gfCNCPoint3[18033] = {X 35.8445, Y 45.9080, Z -4.6667, A 0.000, B 0.000, C 0.000 }
gfCNCPoint3[18034] = {X 35.7593, Y 45.0000, Z -4.6667, A 0.000, B 0.000, C 0.000 }
gfCNCPoint3[18035] = {X 35.7593, Y 44.7148, Z -4.6667, A 0.000, B 0.000, C 0.000 }
gfCNCPoint3[18036] = {X 36.2393, Y 44.7148, Z -4.6667, A 0.000, B 0.000, C 0.000 }
gfCNCPoint3[18037] = {X 36.2397, Y 44.1483, Z -4.6667, A 0.000, B 0.000, C 0.000 }
gfCNCPoint3[18038] = {X 36.3680, Y 43.1522, Z -4.6667, A 0.000, B 0.000, C 0.000 }
gfCNCPoint3[18039] = {X 36.7189, Y 42.2112, Z -4.6667, A 0.000, B 0.000, C 0.000 }
gfCNCPoint3[18040] = {X 37.2740, Y 41.3742, Z -4.6667, A 0.000, B 0.000, C 0.000 }
gfCNCPoint3[18041] = {X 38.0044, Y 40.6849, Z -4.6667, A 0.000, B 0.000, C 0.000 }
gfCNCPoint3[18042] = {X 38.8721, Y 40.1793, Z -4.6667, A 0.000, B 0.000, C 0.000 }
gfCNCPoint3[18043] = {X 39.4558, Y 38.7988, Z -4.6667, A 0.000, B 0.000, C 0.000 }
gfCNCPoint3[18044] = {X 39.9904, Y 37.3987, Z -4.6667, A 0.000, B 0.000, C 0.000 }
gfCNCPoint3[18045] = {X 48.2011, Y 15.3544, Z -4.6667, A 0.000, B 0.000, C 0.000 }
gfCNCPoint3[18046] = {X 47.8187, Y 14.6115, Z -4.6667, A 0.000, B 0.000, C 0.000 }
gfCNCPoint3[18047] = {X 47.5835, Y 13.8097, Z -4.6667, A 0.000, B 0.000, C 0.000 }
gfCNCPoint3[18048] = {X 47.5042, Y 12.9779, Z -4.6667, A 0.000, B 0.000, C 0.000 }
gfCNCPoint3[18049] = {X 47.5042, Y 12.1868, Z -4.6667, A 0.000, B 0.000, C 0.000 }
gfCNCPoint3[18050] = {X 47.6145, Y 11.2077, Z -4.6667, A 0.000, B 0.000, C 0.000 }
gfCNCPoint3[18051] = {X 47.9400, Y 10.2777, Z -4.6667, A 0.000, B 0.000, C 0.000 }
gfCNCPoint3[18052] = {X 48.4642, Y 9.4435, Z -4.6667, A 0.000, B 0.000, C 0.000 }
gfCNCPoint3[18053] = {X 49.1609, Y 8.7468, Z -4.6667, A 0.000, B 0.000, C 0.000 }
gfCNCPoint3[18054] = {X 49.9951, Y 8.2226, Z -4.6667, A 0.000, B 0.000, C 0.000 }
gfCNCPoint3[18055] = {X 50.9251, Y 7.8971, Z -4.6667, A 0.000, B 0.000, C 0.000 }
gfCNCPoint3[18056] = {X 51.9042, Y 7.7868, Z -4.6667, A 0.000, B 0.000, C 0.000 }
gfCNCPoint3[18057] = {X 59.6221, Y 7.7868, Z -4.6667, A 0.000, B 0.000, C 0.000 }
gfCNCPoint3[18058] = {X 60.6012, Y 7.8971, Z -4.6667, A 0.000, B 0.000, C 0.000 }
gfCNCPoint3[18059] = {X 61.5312, Y 8.2226, Z -4.6667, A 0.000, B 0.000, C 0.000 }
gfCNCPoint3[18060] = {X 62.3655, Y 8.7468, Z -4.6667, A 0.000, B 0.000, C 0.000 }
gfCNCPoint3[18061] = {X 63.0622, Y 9.4435, Z -4.6667, A 0.000, B 0.000, C 0.000 }
gfCNCPoint3[18062] = {X 63.5864, Y 10.2777, Z -4.6667, A 0.000, B 0.000, C 0.000 }
gfCNCPoint3[18063] = {X 63.9118, Y 11.2077, Z -4.6667, A 0.000, B 0.000, C 0.000 }
gfCNCPoint3[18064] = {X 64.0221, Y 12.1868, Z -4.6667, A 0.000, B 0.000, C 0.000 }
gfCNCPoint3[18065] = {X 64.0219, Y 13.0233, Z -4.6667, A 0.000, B 0.000, C 0.000 }
gfCNCPoint3[18066] = {X 63.9336, Y 13.8563, Z -4.6667, A 0.000, B 0.000, C 0.000 }
gfCNCPoint3[18067] = {X 63.6890, Y 14.6575, Z -4.6667, A 0.000, B 0.000, C 0.000 }
gfCNCPoint3[18068] = {X 63.2970, Y 15.3978, Z -4.6667, A 0.000, B 0.000, C 0.000 }
gfCNCPoint3[18069] = {X 63.5008, Y 15.9354, Z -4.6667, A 0.000, B 0.000, C 0.000 }
gfCNCPoint3[18070] = {X 66.3154, Y 23.4040, Z -4.6667, A 0.000, B 0.000, C 0.000 }
gfCNCPoint3[18071] = {X 72.2844, Y 39.4717, Z -4.6667, A 0.000, B 0.000, C 0.000 }
gfCNCPoint3[18072] = {X 72.5774, Y 40.2087, Z -4.6667, A 0.000, B 0.000, C 0.000 }
gfCNCPoint3[18073] = {X 73.4349, Y 40.7272, Z -4.6667, A 0.000, B 0.000, C 0.000 }
gfCNCPoint3[18074] = {X 74.1528, Y 41.4262, Z -4.6667, A 0.000, B 0.000, C 0.000 }
gfCNCPoint3[18075] = {X 74.6940, Y 42.2695, Z -4.6667, A 0.000, B 0.000, C 0.000 }
gfCNCPoint3[18076] = {X 75.0304, Y 43.2134, Z -4.6667, A 0.000, B 0.000, C 0.000 }
gfCNCPoint3[18077] = {X 75.1445, Y 44.2089, Z -4.6667, A 0.000, B 0.000, C 0.000 }
gfCNCPoint3[18078] = {X 75.1445, Y 45.0000, Z -4.6667, A 0.000, B 0.000, C 0.000 }
gfCNCPoint3[18079] = {X 75.0341, Y 45.9791, Z -4.6667, A 0.000, B 0.000, C 0.000 }
gfCNCPoint3[18080] = {X 74.7087, Y 46.9091, Z -4.6667, A 0.000, B 0.000, C 0.000 }
gfCNCPoint3[18081] = {X 74.1845, Y 47.7434, Z -4.6667, A 0.000, B 0.000, C 0.000 }
gfCNCPoint3[18082] = {X 73.4878, Y 48.4401, Z -4.6667, A 0.000, B 0.000, C 0.000 }
gfCNCPoint3[18083] = {X 72.6535, Y 48.9643, Z -4.6667, A 0.000, B 0.000, C 0.000 }
gfCNCPoint3[18084] = {X 71.7236, Y 49.2897, Z -4.6667, A 0.000, B 0.000, C 0.000 }
gfCNCPoint3[18085] = {X 70.7445, Y 49.4000, Z -4.6667, A 0.000, B 0.000, C 0.000 }
gfCNCPoint3[18086] = {X 64.1851, Y 49.4000, Z -4.6667, A 0.000, B 0.000, C 0.000 }
gfCNCPoint3[18087] = {X 63.2060, Y 49.2897, Z -4.6667, A 0.000, B 0.000, C 0.000 }
gfCNCPoint3[18088] = {X 62.2760, Y 48.9643, Z -4.6667, A 0.000, B 0.000, C 0.000 }
gfCNCPoint3[18089] = {X 61.4418, Y 48.4401, Z -4.6667, A 0.000, B 0.000, C 0.000 }
gfCNCPoint3[18090] = {X 60.7451, Y 47.7434, Z -4.6667, A 0.000, B 0.000, C 0.000 }
gfCNCPoint3[18091] = {X 60.2209, Y 46.9091, Z -4.6667, A 0.000, B 0.000, C 0.000 }
gfCNCPoint3[18092] = {X 59.8955, Y 45.9791, Z -4.6667, A 0.000, B 0.000, C 0.000 }
gfCNCPoint3[18093] = {X 59.7851, Y 45.0000, Z -4.6667, A 0.000, B 0.000, C 0.000 }
gfCNCPoint3[18094] = {X 59.7856, Y 44.1483, Z -4.6667, A 0.000, B 0.000, C 0.000 }
gfCNCPoint3[18095] = {X 59.8784, Y 43.3079, Z -4.6667, A 0.000, B 0.000, C 0.000 }
gfCNCPoint3[18096] = {X 60.1302, Y 42.5007, Z -4.6667, A 0.000, B 0.000, C 0.000 }
gfCNCPoint3[18097] = {X 60.5318, Y 41.7567, Z -4.6667, A 0.000, B 0.000, C 0.000 }
gfCNCPoint3[18098] = {X 59.9510, Y 40.1692, Z -4.6667, A 0.000, B 0.000, C 0.000 }
gfCNCPoint3[18099] = {X 52.1329, Y 40.1692, Z -4.6667, A 0.000, B 0.000, C 0.000 }
gfCNCPoint3[18100] = {X 51.4225, Y 42.0778, Z -4.6667, A 0.000, B 0.000, C 0.000 }
gfCNCPoint3[18101] = {X 51.7254, Y 42.7537, Z -4.6667, A 0.000, B 0.000, C 0.000 }
gfCNCPoint3[18102] = {X 51.9106, Y 43.4709, Z -4.6667, A 0.000, B 0.000, C 0.000 }
gfCNCPoint3[18103] = {X 51.9729, Y 44.2089, Z -4.6667, A 0.000, B 0.000, C 0.000 }
gfCNCPoint3[18104] = {X 51.9729, Y 45.0000, Z -4.6667, A 0.000, B 0.000, C 0.000 }
gfCNCPoint3[18105] = {X 51.8626, Y 45.9791, Z -4.6667, A 0.000, B 0.000, C 0.000 }
gfCNCPoint3[18106] = {X 51.5372, Y 46.9091, Z -4.6667, A 0.000, B 0.000, C 0.000 }
gfCNCPoint3[18107] = {X 51.0130, Y 47.7434, Z -4.6667, A 0.000, B 0.000, C 0.000 }
gfCNCPoint3[18108] = {X 50.3163, Y 48.4401, Z -4.6667, A 0.000, B 0.000, C 0.000 }
gfCNCPoint3[18109] = {X 49.4820, Y 48.9643, Z -4.6667, A 0.000, B 0.000, C 0.000 }
gfCNCPoint3[18110] = {X 48.5520, Y 49.2897, Z -4.6667, A 0.000, B 0.000, C 0.000 }
gfCNCPoint3[18111] = {X 47.5729, Y 49.4000, Z -4.6667, A 0.000, B 0.000, C 0.000 }
gfCNCPoint3[18112] = {X 40.6393, Y 49.4000, Z -4.6667, A 0.000, B 0.000, C 0.000 }
gfCNCPoint3[18113] = {X 39.6602, Y 49.2897, Z -4.6667, A 0.000, B 0.000, C 0.000 }
gfCNCPoint3[18114] = {X 38.7302, Y 48.9643, Z -4.6667, A 0.000, B 0.000, C 0.000 }
gfCNCPoint3[18115] = {X 37.8959, Y 48.4401, Z -4.6667, A 0.000, B 0.000, C 0.000 }
gfCNCPoint3[18116] = {X 37.1992, Y 47.7434, Z -4.6667, A 0.000, B 0.000, C 0.000 }
gfCNCPoint3[18117] = {X 36.6750, Y 46.9091, Z -4.6667, A 0.000, B 0.000, C 0.000 }
gfCNCPoint3[18118] = {X 36.3496, Y 45.9791, Z -4.6667, A 0.000, B 0.000, C 0.000 }
gfCNCPoint3[18119] = {X 36.2393, Y 45.0000, Z -4.6667, A 0.000, B 0.000, C 0.000 }
gfCNCPoint3[18120] = {X 36.2393, Y 44.7148, Z -4.6667, A 0.000, B 0.000, C 0.000 }
gfCNCPoint3[18121] = {X 35.7593, Y 44.7148, Z -4.6667, A 0.000, B 0.000, C 0.000 }
gfCNCPoint3[18122] = {X 35.2211, Y 46.0074, Z -4.6667, A 0.000, B 0.000, C 0.000 }
gfCNCPoint3[18123] = {X 34.4930, Y 47.2034, Z -4.6667, A 0.000, B 0.000, C 0.000 }
gfCNCPoint3[18124] = {X 33.5918, Y 48.2750, Z -4.6667, A 0.000, B 0.000, C 0.000 }
gfCNCPoint3[18125] = {X 33.2092, Y 48.6435, Z -4.6667, A 0.000, B 0.000, C 0.000 }
gfCNCPoint3[18126] = {X 32.8060, Y 48.9892, Z -4.6667, A 0.000, B 0.000, C 0.000 }
gfCNCPoint3[18127] = {X 32.2679, Y 49.4243, Z -4.6667, A 0.000, B 0.000, C 0.000 }
gfCNCPoint3[18128] = {X 31.1814, Y 50.1797, Z -4.6667, A 0.000, B 0.000, C 0.000 }
gfCNCPoint3[18129] = {X 29.9980, Y 50.7716, Z -4.6667, A 0.000, B 0.000, C 0.000 }
gfCNCPoint3[18130] = {X 28.7420, Y 51.1880, Z -4.6667, A 0.000, B 0.000, C 0.000 }
gfCNCPoint3[18131] = {X 27.4393, Y 51.4201, Z -4.6667, A 0.000, B 0.000, C 0.000 }
gfCNCPoint3[18132] = {X 26.1168, Y 51.4633, Z -4.6667, A 0.000, B 0.000, C 0.000 }
gfCNCPoint3[18133] = {X 23.6796, Y 52.5818, Z -4.6667, A 0.000, B 0.000, C 0.000 }
gfCNCPoint3[18134] = {X 21.1619, Y 53.5051, Z -4.6667, A 0.000, B 0.000, C 0.000 }
gfCNCPoint3[18135] = {X 18.9497, Y 54.1342, Z -4.6667, A 0.000, B 0.000, C 0.000 }
gfCNCPoint3[18136] = {X 16.6929, Y 54.5773, Z -4.6667, A 0.000, B 0.000, C 0.000 }
gfCNCPoint3[18137] = {X 14.4071, Y 54.8314, Z -4.6667, A 0.000, B 0.000, C 0.000 }
gfCNCPoint3[18138] = {X 12.1081, Y 54.8947, Z -4.6667, A 0.000, B 0.000, C 0.000 }
gfCNCPoint3[18139] = {X 9.8118, Y 54.7667, Z -4.6667, A 0.000, B 0.000, C 0.000 }
gfCNCPoint3[18140] = {X 7.5341, Y 54.4485, Z -4.6667, A 0.000, B 0.000, C 0.000 }
gfCNCPoint3[18141] = {X 7.1099, Y 54.3677, Z -4.6667, A 0.000, B 0.000, C 0.000 }
gfCNCPoint3[18142] = {X 6.6870, Y 54.2803, Z -4.6667, A 0.000, B 0.000, C 0.000 }
gfCNCPoint3[18143] = {X 5.6890, Y 54.0441, Z -4.6667, A 0.000, B 0.000, C 0.000 }
gfCNCPoint3[18144] = {X 4.7034, Y 53.7607, Z -4.6667, A 0.000, B 0.000, C 0.000 }
gfCNCPoint3[18145] = {X 4.7034, Y 95.2950, Z -4.6667, A 0.000, B 0.000, C 0.000 }
gfCNCPoint3[18146] = {X 117.9387, Y 95.2950, Z -4.6667, A 0.000, B 0.000, C 0.000 }
gfCNCPoint3[18147] = {X 118.3612, Y 94.0786, Z -4.6667, A 0.000, B 0.000, C 0.000 }
gfCNCPoint3[18148] = {X 118.9914, Y 92.9556, Z -4.6667, A 0.000, B 0.000, C 0.000 }
gfCNCPoint3[18149] = {X 119.8096, Y 91.9613, Z -4.6667, A 0.000, B 0.000, C 0.000 }
gfCNCPoint3[18150] = {X 120.7902, Y 91.1266, Z -4.6667, A 0.000, B 0.000, C 0.000 }
gfCNCPoint3[18151] = {X 121.9025, Y 90.4778, Z -4.6667, A 0.000, B 0.000, C 0.000 }
gfCNCPoint3[18152] = {X 123.1117, Y 90.0351, Z -4.6667, A 0.000, B 0.000, C 0.000 }
gfCNCPoint3[18153] = {X 124.3800, Y 89.8124, Z -4.6667, A 0.000, B 0.000, C 0.000 }
gfCNCPoint3[18154] = {X 125.0501, Y 89.7112, Z -4.6667, A 0.000, B 0.000, C 0.000 }
gfCNCPoint3[18155] = {X 125.3582, Y 89.6652, Z -4.6667, A 0.000, B 0.000, C 0.000 }
gfCNCPoint3[18156] = {X 125.6646, Y 89.6090, Z -4.6667, A 0.000, B 0.000, C 0.000 }
gfCNCPoint3[18157] = {X 126.4915, Y 88.7984, Z -4.6667, A 0.000, B 0.000, C 0.000 }
gfCNCPoint3[18158] = {X 127.2841, Y 87.9542, Z -4.6667, A 0.000, B 0.000, C 0.000 }
gfCNCPoint3[18159] = {X 152.2076, Y 60.5847, Z -4.6667, A 0.000, B 0.000, C 0.000 }
gfCNCPoint3[18160] = {X 152.0684, Y 59.7898, Z -4.6667, A 0.000, B 0.000, C 0.000 }
gfCNCPoint3[18161] = {X 152.0181, Y 58.9845, Z -4.6667, A 0.000, B 0.000, C 0.000 }
gfCNCPoint3[18162] = {X 152.0180, Y 58.0000, Z -4.6667, A 0.000, B 0.000, C 0.000 }
gfCNCPoint3[18163] = {X 152.1286, Y 56.7358, Z -4.6667, A 0.000, B 0.000, C 0.000 }
gfCNCPoint3[18164] = {X 152.4570, Y 55.5101, Z -4.6667, A 0.000, B 0.000, C 0.000 }
gfCNCPoint3[18165] = {X 152.9933, Y 54.3600, Z -4.6667, A 0.000, B 0.000, C 0.000 }
gfCNCPoint3[18166] = {X 153.7212, Y 53.3205, Z -4.6667, A 0.000, B 0.000, C 0.000 }
gfCNCPoint3[18167] = {X 154.6185, Y 52.4232, Z -4.6667, A 0.000, B 0.000, C 0.000 }
gfCNCPoint3[18168] = {X 155.6580, Y 51.6953, Z -4.6667, A 0.000, B 0.000, C 0.000 }
gfCNCPoint3[18169] = {X 156.8081, Y 51.1590, Z -4.6667, A 0.000, B 0.000, C 0.000 }
gfCNCPoint3[18170] = {X 158.0338, Y 50.8306, Z -4.6667, A 0.000, B 0.000, C 0.000 }
gfCNCPoint3[18171] = {X 159.2980, Y 50.7200, Z -4.6667, A 0.000, B 0.000, C 0.000 }
gfCNCPoint3[18172] = {X 178.5335, Y 50.7200, Z -4.6667, A 0.000, B 0.000, C 0.000 }
gfCNCPoint3[18173] = {X 179.7870, Y 50.8287, Z -4.6667, A 0.000, B 0.000, C 0.000 }
gfCNCPoint3[18174] = {X 181.0031, Y 51.1517, Z -4.6667, A 0.000, B 0.000, C 0.000 }
gfCNCPoint3[18175] = {X 182.1454, Y 51.6792, Z -4.6667, A 0.000, B 0.000, C 0.000 }
gfCNCPoint3[18176] = {X 183.1798, Y 52.3955, Z -4.6667, A 0.000, B 0.000, C 0.000 }
gfCNCPoint3[18177] = {X 184.0880, Y 53.2941, Z -4.6667, A 0.000, B 0.000, C 0.000 }
gfCNCPoint3[18178] = {X 184.8252, Y 54.3376, Z -4.6667, A 0.000, B 0.000, C 0.000 }
gfCNCPoint3[18179] = {X 185.3685, Y 55.4939, Z -4.6667, A 0.000, B 0.000, C 0.000 }
gfCNCPoint3[18180] = {X 185.7014, Y 56.7273, Z -4.6667, A 0.000, B 0.000, C 0.000 }
gfCNCPoint3[18181] = {X 185.8135, Y 58.0000, Z -4.6667, A 0.000, B 0.000, C 0.000 }
gfCNCPoint3[18182] = {X 185.8133, Y 58.9942, Z -4.6667, A 0.000, B 0.000, C 0.000 }
gfCNCPoint3[18183] = {X 185.7648, Y 59.7749, Z -4.6667, A 0.000, B 0.000, C 0.000 }
gfCNCPoint3[18184] = {X 185.6328, Y 60.5459, Z -4.6667, A 0.000, B 0.000, C 0.000 }
gfCNCPoint3[18185] = {X 211.6613, Y 88.9545, Z -4.6667, A 0.000, B 0.000, C 0.000 }
gfCNCPoint3[18186] = {X 212.0333, Y 89.3391, Z -4.6667, A 0.000, B 0.000, C 0.000 }
gfCNCPoint3[18187] = {X 212.4256, Y 89.7031, Z -4.6667, A 0.000, B 0.000, C 0.000 }
gfCNCPoint3[18188] = {X 212.6034, Y 89.7411, Z -4.6667, A 0.000, B 0.000, C 0.000 }
gfCNCPoint3[18189] = {X 213.4473, Y 89.8474, Z -4.6667, A 0.000, B 0.000, C 0.000 }
gfCNCPoint3[18190] = {X 214.4298, Y 89.7705, Z -4.6667, A 0.000, B 0.000, C 0.000 }
gfCNCPoint3[18191] = {X 215.4138, Y 89.7168, Z -4.6667, A 0.000, B 0.000, C 0.000 }
gfCNCPoint3[18192] = {X 215.6261, Y 89.6935, Z -4.6667, A 0.000, B 0.000, C 0.000 }
gfCNCPoint3[18193] = {X 215.8213, Y 89.6066, Z -4.6667, A 0.000, B 0.000, C 0.000 }
gfCNCPoint3[18194] = {X 239.3462, Y 74.5356, Z -4.6667, A 0.000, B 0.000, C 0.000 }
gfCNCPoint3[18195] = {X 220.5436, Y 67.1569, Z -4.6667, A 0.000, B 0.000, C 0.000 }
gfCNCPoint3[18196] = {X 219.0950, Y 66.6707, Z -4.6667, A 0.000, B 0.000, C 0.000 }
gfCNCPoint3[18197] = {X 217.6003, Y 66.3535, Z -4.6667, A 0.000, B 0.000, C 0.000 }
gfCNCPoint3[18198] = {X 216.0790, Y 66.2097, Z -4.6667, A 0.000, B 0.000, C 0.000 }
gfCNCPoint3[18199] = {X 214.8523, Y 66.0623, Z -4.6667, A 0.000, B 0.000, C 0.000 }
gfCNCPoint3[18200] = {X 213.6682, Y 65.7097, Z -4.6667, A 0.000, B 0.000, C 0.000 }
gfCNCPoint3[18201] = {X 212.5607, Y 65.1618, Z -4.6667, A 0.000, B 0.000, C 0.000 }
gfCNCPoint3[18202] = {X 211.5619, Y 64.4346, Z -4.6667, A 0.000, B 0.000, C 0.000 }
gfCNCPoint3[18203] = {X 210.7004, Y 63.5490, Z -4.6667, A 0.000, B 0.000, C 0.000 }
gfCNCPoint3[18204] = {X 210.0011, Y 62.5304, Z -4.6667, A 0.000, B 0.000, C 0.000 }
gfCNCPoint3[18205] = {X 209.4841, Y 61.4082, Z -4.6667, A 0.000, B 0.000, C 0.000 }
gfCNCPoint3[18206] = {X 209.1643, Y 60.2148, Z -4.6667, A 0.000, B 0.000, C 0.000 }
gfCNCPoint3[18207] = {X 209.0510, Y 58.9845, Z -4.6667, A 0.000, B 0.000, C 0.000 }
gfCNCPoint3[18208] = {X 209.0508, Y 58.0000, Z -4.6667, A 0.000, B 0.000, C 0.000 }
gfCNCPoint3[18209] = {X 209.1477, Y 56.8162, Z -4.6667, A 0.000, B 0.000, C 0.000 }
gfCNCPoint3[18210] = {X 209.4358, Y 55.6638, Z -4.6667, A 0.000, B 0.000, C 0.000 }
gfCNCPoint3[18211] = {X 209.9075, Y 54.5737, Z -4.6667, A 0.000, B 0.000, C 0.000 }
gfCNCPoint3[18212] = {X 210.5502, Y 53.5748, Z -4.6667, A 0.000, B 0.000, C 0.000 }
gfCNCPoint3[18213] = {X 211.3467, Y 52.6937, Z -4.6667, A 0.000, B 0.000, C 0.000 }
gfCNCPoint3[18214] = {X 212.2759, Y 51.9538, Z -4.6667, A 0.000, B 0.000, C 0.000 }
gfCNCPoint3[18215] = {X 213.3131, Y 51.3749, Z -4.6667, A 0.000, B 0.000, C 0.000 }
gfCNCPoint3[18216] = {X 214.4306, Y 50.9724, Z -4.6667, A 0.000, B 0.000, C 0.000 }
gfCNCPoint3[18217] = {X 215.3724, Y 50.7834, Z -4.6667, A 0.000, B 0.000, C 0.000 }
gfCNCPoint3[18218] = {X 216.3308, Y 50.7200, Z -4.6667, A 0.000, B 0.000, C 0.000 }
gfCNCPoint3[18219] = {X 237.2617, Y 50.7200, Z -4.6667, A 0.000, B 0.000, C 0.000 }
gfCNCPoint3[18220] = {X 238.3057, Y 50.7953, Z -4.6667, A 0.000, B 0.000, C 0.000 }
gfCNCPoint3[18221] = {X 239.3282, Y 51.0195, Z -4.6667, A 0.000, B 0.000, C 0.000 }
gfCNCPoint3[18222] = {X 240.3080, Y 51.3880, Z -4.6667, A 0.000, B 0.000, C 0.000 }
gfCNCPoint3[18223] = {X 241.2247, Y 51.8932, Z -4.6667, A 0.000, B 0.000, C 0.000 }
gfCNCPoint3[18224] = {X 242.0741, Y 52.5375, Z -4.6667, A 0.000, B 0.000, C 0.000 }
gfCNCPoint3[18225] = {X 242.8203, Y 53.2989, Z -4.6667, A 0.000, B 0.000, C 0.000 }
gfCNCPoint3[18226] = {X 243.4473, Y 54.1611, Z -4.6667, A 0.000, B 0.000, C 0.000 }
gfCNCPoint3[18227] = {X 243.9416, Y 55.1057, Z -4.6667, A 0.000, B 0.000, C 0.000 }
gfCNCPoint3[18228] = {X 244.2927, Y 56.1123, Z -4.6667, A 0.000, B 0.000, C 0.000 }
gfCNCPoint3[18229] = {X 249.2034, Y 58.0271, Z -4.6667, A 0.000, B 0.000, C 0.000 }
gfCNCPoint3[18230] = {X 272.6725, Y 67.3425, Z -4.6667, A 0.000, B 0.000, C 0.000 }
gfCNCPoint3[18231] = {X 272.6724, Y 65.2841, Z -4.6667, A 0.000, B 0.000, C 0.000 }
gfCNCPoint3[18232] = {X 271.6649, Y 64.6027, Z -4.6667, A 0.000, B 0.000, C 0.000 }
gfCNCPoint3[18233] = {X 270.7849, Y 63.7631, Z -4.6667, A 0.000, B 0.000, C 0.000 }
gfCNCPoint3[18234] = {X 270.0569, Y 62.7887, Z -4.6667, A 0.000, B 0.000, C 0.000 }
gfCNCPoint3[18235] = {X 269.5014, Y 61.7068, Z -4.6667, A 0.000, B 0.000, C 0.000 }
gfCNCPoint3[18236] = {X 269.2026, Y 60.8253, Z -4.6667, A 0.000, B 0.000, C 0.000 }
gfCNCPoint3[18237] = {X 269.0188, Y 59.9129, Z -4.6667, A 0.000, B 0.000, C 0.000 }
gfCNCPoint3[18238] = {X 268.9529, Y 58.9845, Z -4.6667, A 0.000, B 0.000, C 0.000 }
gfCNCPoint3[18239] = {X 268.9527, Y 58.0000, Z -4.6667, A 0.000, B 0.000, C 0.000 }
gfCNCPoint3[18240] = {X 269.0633, Y 56.7358, Z -4.6667, A 0.000, B 0.000, C 0.000 }
gfCNCPoint3[18241] = {X 269.3917, Y 55.5101, Z -4.6667, A 0.000, B 0.000, C 0.000 }
gfCNCPoint3[18242] = {X 269.9280, Y 54.3600, Z -4.6667, A 0.000, B 0.000, C 0.000 }
gfCNCPoint3[18243] = {X 270.6559, Y 53.3205, Z -4.6667, A 0.000, B 0.000, C 0.000 }
gfCNCPoint3[18244] = {X 271.5532, Y 52.4232, Z -4.6667, A 0.000, B 0.000, C 0.000 }
gfCNCPoint3[18245] = {X 272.5927, Y 51.6953, Z -4.6667, A 0.000, B 0.000, C 0.000 }
gfCNCPoint3[18246] = {X 273.7428, Y 51.1590, Z -4.6667, A 0.000, B 0.000, C 0.000 }
gfCNCPoint3[18247] = {X 274.9685, Y 50.8306, Z -4.6667, A 0.000, B 0.000, C 0.000 }
gfCNCPoint3[18248] = {X 276.2327, Y 50.7200, Z -4.6667, A 0.000, B 0.000, C 0.000 }
gfCNCPoint3[18249] = {X 292.7731, Y 50.7200, Z -4.6667, A 0.000, B 0.000, C 0.000 }
gfCNCPoint3[18250] = {X 293.4209, Y 50.7489, Z -4.6667, A 0.000, B 0.000, C 0.000 }
gfCNCPoint3[18251] = {X 294.0636, Y 50.8353, Z -4.6667, A 0.000, B 0.000, C 0.000 }
gfCNCPoint3[18252] = {X 294.7294, Y 50.9878, Z -4.6667, A 0.000, B 0.000, C 0.000 }
gfCNCPoint3[18253] = {X 295.3780, Y 51.2020, Z -4.6667, A 0.000, B 0.000, C 0.000 }
gfCNCPoint3[18254] = {X 298.3089, Y 43.5533, Z -4.6667, A 0.000, B 0.000, C 0.000 }
gfCNCPoint3[18255] = {X 298.4821, Y 42.5299, Z -4.6667, A 0.000, B 0.000, C 0.000 }
gfCNCPoint3[18256] = {X 298.7926, Y 41.5395, Z -4.6667, A 0.000, B 0.000, C 0.000 }
gfCNCPoint3[18257] = {X 299.2345, Y 40.6003, Z -4.6667, A 0.000, B 0.000, C 0.000 }
gfCNCPoint3[18258] = {X 299.7997, Y 39.7298, Z -4.6667, A 0.000, B 0.000, C 0.000 }
gfCNCPoint3[18259] = {X 299.7997, Y 36.9943, Z -4.6667, A 0.000, B 0.000, C 0.000 }
gfCNCPoint3[18260] = {X 296.8141, Y 36.9943, Z -4.6667, A 0.000, B 0.000, C 0.000 }
gfCNCPoint3[18261] = {X 296.8138, Y 39.7485, Z -4.6667, A 0.000, B 0.000, C 0.000 }
gfCNCPoint3[18262] = {X 297.3851, Y 40.6112, Z -4.6667, A 0.000, B 0.000, C 0.000 }
gfCNCPoint3[18263] = {X 297.8301, Y 41.5453, Z -4.6667, A 0.000, B 0.000, C 0.000 }
gfCNCPoint3[18264] = {X 298.1401, Y 42.5325, Z -4.6667, A 0.000, B 0.000, C 0.000 }
gfCNCPoint3[18265] = {X 298.3089, Y 43.5533, Z -4.6667, A 0.000, B 0.000, C 0.000 }
gfCNCPoint3[18266] = {X 296.2368, Y 48.9609, Z -4.6667, A 0.000, B 0.000, C 0.000 }
gfCNCPoint3[18267] = {X 296.6126, Y 49.1140, Z -4.6667, A 0.000, B 0.000, C 0.000 }
gfCNCPoint3[18268] = {X 296.9817, Y 49.2828, Z -4.6667, A 0.000, B 0.000, C 0.000 }
gfCNCPoint3[18269] = {X 297.2571, Y 49.4212, Z -4.6667, A 0.000, B 0.000, C 0.000 }
gfCNCPoint3[18270] = {X 297.5280, Y 49.5683, Z -4.6667, A 0.000, B 0.000, C 0.000 }
gfCNCPoint3[18271] = {X 298.7174, Y 50.3602, Z -4.6667, A 0.000, B 0.000, C 0.000 }
gfCNCPoint3[18272] = {X 299.7774, Y 51.3185, Z -4.6667, A 0.000, B 0.000, C 0.000 }
gfCNCPoint3[18273] = {X 300.6847, Y 52.4224, Z -4.6667, A 0.000, B 0.000, C 0.000 }
gfCNCPoint3[18274] = {X 301.5914, Y 51.3191, Z -4.6667, A 0.000, B 0.000, C 0.000 }
gfCNCPoint3[18275] = {X 302.6506, Y 50.3611, Z -4.6667, A 0.000, B 0.000, C 0.000 }
gfCNCPoint3[18276] = {X 303.8393, Y 49.5695, Z -4.6667, A 0.000, B 0.000, C 0.000 }
gfCNCPoint3[18277] = {X 302.8989, Y 49.0956, Z -4.6667, A 0.000, B 0.000, C 0.000 }
gfCNCPoint3[18278] = {X 302.0820, Y 48.4310, Z -4.6667, A 0.000, B 0.000, C 0.000 }
gfCNCPoint3[18279] = {X 301.4268, Y 47.6067, Z -4.6667, A 0.000, B 0.000, C 0.000 }
gfCNCPoint3[18280] = {X 300.9636, Y 46.6610, Z -4.6667, A 0.000, B 0.000, C 0.000 }
gfCNCPoint3[18281] = {X 300.7923, Y 46.0759, Z -4.6667, A 0.000, B 0.000, C 0.000 }
gfCNCPoint3[18282] = {X 300.6953, Y 45.4741, Z -4.6667, A 0.000, B 0.000, C 0.000 }
gfCNCPoint3[18283] = {X 300.6790, Y 45.2570, Z -4.6667, A 0.000, B 0.000, C 0.000 }
gfCNCPoint3[18284] = {X 300.6724, Y 45.0393, Z -4.6667, A 0.000, B 0.000, C 0.000 }
gfCNCPoint3[18285] = {X 300.6725, Y 44.1879, Z -4.6667, A 0.000, B 0.000, C 0.000 }
gfCNCPoint3[18286] = {X 300.6810, Y 43.9898, Z -4.6667, A 0.000, B 0.000, C 0.000 }
gfCNCPoint3[18287] = {X 300.6970, Y 43.7921, Z -4.6667, A 0.000, B 0.000, C 0.000 }
gfCNCPoint3[18288] = {X 300.8618, Y 42.9127, Z -4.6667, A 0.000, B 0.000, C 0.000 }
gfCNCPoint3[18289] = {X 301.1739, Y 42.0742, Z -4.6667, A 0.000, B 0.000, C 0.000 }
gfCNCPoint3[18290] = {X 301.6243, Y 41.3011, Z -4.6667, A 0.000, B 0.000, C 0.000 }
gfCNCPoint3[18291] = {X 302.1997, Y 40.6160, Z -4.6667, A 0.000, B 0.000, C 0.000 }
gfCNCPoint3[18292] = {X 302.1997, Y 34.5943, Z -4.6667, A 0.000, B 0.000, C 0.000 }
gfCNCPoint3[18293] = {X 294.4144, Y 34.5943, Z -4.6667, A 0.000, B 0.000, C 0.000 }
gfCNCPoint3[18294] = {X 294.4137, Y 40.6555, Z -4.6667, A 0.000, B 0.000, C 0.000 }
gfCNCPoint3[18295] = {X 294.9940, Y 41.3224, Z -4.6667, A 0.000, B 0.000, C 0.000 }
gfCNCPoint3[18296] = {X 295.4471, Y 42.0814, Z -4.6667, A 0.000, B 0.000, C 0.000 }
gfCNCPoint3[18297] = {X 295.7589, Y 42.9086, Z -4.6667, A 0.000, B 0.000, C 0.000 }
gfCNCPoint3[18298] = {X 295.9194, Y 43.7779, Z -4.6667, A 0.000, B 0.000, C 0.000 }
gfCNCPoint3[18299] = {X 295.9349, Y 43.9931, Z -4.6667, A 0.000, B 0.000, C 0.000 }
gfCNCPoint3[18300] = {X 295.9411, Y 44.2089, Z -4.6667, A 0.000, B 0.000, C 0.000 }
gfCNCPoint3[18301] = {X 295.9411, Y 45.0000, Z -4.6667, A 0.000, B 0.000, C 0.000 }
gfCNCPoint3[18302] = {X 295.9354, Y 45.2373, Z -4.6667, A 0.000, B 0.000, C 0.000 }
gfCNCPoint3[18303] = {X 295.9181, Y 45.4741, Z -4.6667, A 0.000, B 0.000, C 0.000 }
gfCNCPoint3[18304] = {X 298.3067, Y 45.7073, Z -4.6667, A 0.000, B 0.000, C 0.000 }
gfCNCPoint3[18305] = {X 298.2010, Y 46.4214, Z -4.6667, A 0.000, B 0.000, C 0.000 }
gfCNCPoint3[18306] = {X 298.0252, Y 47.1215, Z -4.6667, A 0.000, B 0.000, C 0.000 }
gfCNCPoint3[18307] = {X 298.3689, Y 47.2942, Z -4.6667, A 0.000, B 0.000, C 0.000 }
gfCNCPoint3[18308] = {X 298.7069, Y 47.4778, Z -4.6667, A 0.000, B 0.000, C 0.000 }
gfCNCPoint3[18309] = {X 298.4514, Y 46.6051, Z -4.6667, A 0.000, B 0.000, C 0.000 }
gfCNCPoint3[18310] = {X 298.3067, Y 45.7073, Z -4.6667, A 0.000, B 0.000, C 0.000 }
gfCNCPoint3[18311] = {X 295.9181, Y 45.4741, Z -4.6667, A 0.000, B 0.000, C 0.000 }
gfCNCPoint3[18312] = {X 295.8472, Y 45.9528, Z -4.6667, A 0.000, B 0.000, C 0.000 }
gfCNCPoint3[18313] = {X 295.7293, Y 46.4221, Z -4.6667, A 0.000, B 0.000, C 0.000 }
gfCNCPoint3[18314] = {X 295.4314, Y 47.1714, Z -4.6667, A 0.000, B 0.000, C 0.000 }
gfCNCPoint3[18315] = {X 295.0142, Y 47.8614, Z -4.6667, A 0.000, B 0.000, C 0.000 }
gfCNCPoint3[18316] = {X 294.4890, Y 48.4733, Z -4.6667, A 0.000, B 0.000, C 0.000 }
gfCNCPoint3[18317] = {X 295.3744, Y 48.6761, Z -4.6667, A 0.000, B 0.000, C 0.000 }
gfCNCPoint3[18318] = {X 296.2368, Y 48.9609, Z -4.6667, A 0.000, B 0.000, C 0.000 }
gfCNCPoint3[18319] = {X 295.3780, Y 51.2020, Z -4.6667, A 0.000, B 0.000, C 0.000 }
gfCNCPoint3[18320] = {X 296.3501, Y 51.6594, Z -4.6667, A 0.000, B 0.000, C 0.000 }
gfCNCPoint3[18321] = {X 297.2442, Y 52.2548, Z -4.6667, A 0.000, B 0.000, C 0.000 }
gfCNCPoint3[18322] = {X 298.0410, Y 52.9753, Z -4.6667, A 0.000, B 0.000, C 0.000 }
gfCNCPoint3[18323] = {X 298.7231, Y 53.8053, Z -4.6667, A 0.000, B 0.000, C 0.000 }
gfCNCPoint3[18324] = {X 299.2946, Y 54.7645, Z -4.6667, A 0.000, B 0.000, C 0.000 }
gfCNCPoint3[18325] = {X 299.7126, Y 55.7997, Z -4.6667, A 0.000, B 0.000, C 0.000 }
gfCNCPoint3[18326] = {X 299.9675, Y 56.8868, Z -4.6667, A 0.000, B 0.000, C 0.000 }
gfCNCPoint3[18327] = {X 300.0531, Y 58.0000, Z -4.6667, A 0.000, B 0.000, C 0.000 }
gfCNCPoint3[18328] = {X 300.0531, Y 58.9443, Z -4.6667, A 0.000, B 0.000, C 0.000 }
gfCNCPoint3[18329] = {X 299.9647, Y 60.0540, Z -4.6667, A 0.000, B 0.000, C 0.000 }
gfCNCPoint3[18330] = {X 299.7085, Y 61.1374, Z -4.6667, A 0.000, B 0.000, C 0.000 }
gfCNCPoint3[18331] = {X 299.2905, Y 62.1692, Z -4.6667, A 0.000, B 0.000, C 0.000 }
gfCNCPoint3[18332] = {X 298.7205, Y 63.1253, Z -4.6667, A 0.000, B 0.000, C 0.000 }
gfCNCPoint3[18333] = {X 300.6821, Y 64.5080, Z -4.6667, A 0.000, B 0.000, C 0.000 }
gfCNCPoint3[18334] = {X 299.7826, Y 65.6042, Z -4.6667, A 0.000, B 0.000, C 0.000 }
gfCNCPoint3[18335] = {X 298.7328, Y 66.5575, Z -4.6667, A 0.000, B 0.000, C 0.000 }
gfCNCPoint3[18336] = {X 298.7328, Y 89.4421, Z -4.6667, A 0.000, B 0.000, C 0.000 }
gfCNCPoint3[18337] = {X 299.8295, Y 90.4465, Z -4.6667, A 0.000, B 0.000, C 0.000 }
gfCNCPoint3[18338] = {X 300.7599, Y 91.6065, Z -4.6667, A 0.000, B 0.000, C 0.000 }
gfCNCPoint3[18339] = {X 301.5024, Y 92.8950, Z -4.6667, A 0.000, B 0.000, C 0.000 }
gfCNCPoint3[18340] = {X 304.0672, Y 92.8950, Z -4.6667, A 0.000, B 0.000, C 0.000 }
gfCNCPoint3[18341] = {X 303.7096, Y 91.9001, Z -4.6667, A 0.000, B 0.000, C 0.000 }
gfCNCPoint3[18342] = {X 303.4136, Y 90.8851, Z -4.6667, A 0.000, B 0.000, C 0.000 }
gfCNCPoint3[18343] = {X 302.9745, Y 88.8145, Z -4.6667, A 0.000, B 0.000, C 0.000 }
gfCNCPoint3[18344] = {X 302.7144, Y 86.7139, Z -4.6667, A 0.000, B 0.000, C 0.000 }
gfCNCPoint3[18345] = {X 302.6354, Y 84.5987, Z -4.6667, A 0.000, B 0.000, C 0.000 }
gfCNCPoint3[18346] = {X 302.6364, Y 66.5619, Z -4.6667, A 0.000, B 0.000, C 0.000 }
gfCNCPoint3[18347] = {X 301.5837, Y 65.6069, Z -4.6667, A 0.000, B 0.000, C 0.000 }
gfCNCPoint3[18348] = {X 300.6821, Y 64.5080, Z -4.6667, A 0.000, B 0.000, C 0.000 }
gfCNCPoint3[18349] = {X 298.7205, Y 63.1253, Z -4.6667, A 0.000, B 0.000, C 0.000 }
gfCNCPoint3[18350] = {X 298.0344, Y 63.9598, Z -4.6667, A 0.000, B 0.000, C 0.000 }
gfCNCPoint3[18351] = {X 297.2326, Y 64.6839, Z -4.6667, A 0.000, B 0.000, C 0.000 }
gfCNCPoint3[18352] = {X 296.3328, Y 65.2816, Z -4.6667, A 0.000, B 0.000, C 0.000 }
gfCNCPoint3[18353] = {X 296.3328, Y 90.7164, Z -4.6667, A 0.000, B 0.000, C 0.000 }
gfCNCPoint3[18354] = {X 297.3129, Y 91.3791, Z -4.6667, A 0.000, B 0.000, C 0.000 }
gfCNCPoint3[18355] = {X 298.1734, Y 92.1912, Z -4.6667, A 0.000, B 0.000, C 0.000 }
gfCNCPoint3[18356] = {X 298.8916, Y 93.1314, Z -4.6667, A 0.000, B 0.000, C 0.000 }
gfCNCPoint3[18357] = {X 299.4488, Y 94.1751, Z -4.6667, A 0.000, B 0.000, C 0.000 }
gfCNCPoint3[18358] = {X 299.8304, Y 95.2950, Z -4.6667, A 0.000, B 0.000, C 0.000 }
gfCNCPoint3[18359] = {X 308.0991, Y 95.2950, Z -4.6667, A 0.000, B 0.000, C 0.000 }
gfCNCPoint3[18360] = {X 307.0960, Y 93.7116, Z -4.6667, A 0.000, B 0.000, C 0.000 }
gfCNCPoint3[18361] = {X 306.2999, Y 92.0146, Z -4.6667, A 0.000, B 0.000, C 0.000 }
gfCNCPoint3[18362] = {X 305.9920, Y 91.1578, Z -4.6667, A 0.000, B 0.000, C 0.000 }
gfCNCPoint3[18363] = {X 305.7370, Y 90.2838, Z -4.6667, A 0.000, B 0.000, C 0.000 }
gfCNCPoint3[18364] = {X 305.3407, Y 88.4136, Z -4.6667, A 0.000, B 0.000, C 0.000 }
gfCNCPoint3[18365] = {X 305.1063, Y 86.5162, Z -4.6667, A 0.000, B 0.000, C 0.000 }
gfCNCPoint3[18366] = {X 305.0354, Y 84.6057, Z -4.6667, A 0.000, B 0.000, C 0.000 }
gfCNCPoint3[18367] = {X 305.0365, Y 65.2844, Z -4.6667, A 0.000, B 0.000, C 0.000 }
gfCNCPoint3[18368] = {X 304.1346, Y 64.6867, Z -4.6667, A 0.000, B 0.000, C 0.000 }
gfCNCPoint3[18369] = {X 303.3313, Y 63.9619, Z -4.6667, A 0.000, B 0.000, C 0.000 }
gfCNCPoint3[18370] = {X 302.6443, Y 63.1261, Z -4.6667, A 0.000, B 0.000, C 0.000 }
gfCNCPoint3[18371] = {X 302.0792, Y 62.1787, Z -4.6667, A 0.000, B 0.000, C 0.000 }
gfCNCPoint3[18372] = {X 301.6638, Y 61.1568, Z -4.6667, A 0.000, B 0.000, C 0.000 }
gfCNCPoint3[18373] = {X 301.4076, Y 60.0838, Z -4.6667, A 0.000, B 0.000, C 0.000 }
gfCNCPoint3[18374] = {X 301.3164, Y 58.9845, Z -4.6667, A 0.000, B 0.000, C 0.000 }
gfCNCPoint3[18375] = {X 301.3162, Y 58.0000, Z -4.6667, A 0.000, B 0.000, C 0.000 }
gfCNCPoint3[18376] = {X 301.4018, Y 56.8868, Z -4.6667, A 0.000, B 0.000, C 0.000 }
gfCNCPoint3[18377] = {X 301.6567, Y 55.7997, Z -4.6667, A 0.000, B 0.000, C 0.000 }
gfCNCPoint3[18378] = {X 302.0747, Y 54.7645, Z -4.6667, A 0.000, B 0.000, C 0.000 }
gfCNCPoint3[18379] = {X 302.6462, Y 53.8053, Z -4.6667, A 0.000, B 0.000, C 0.000 }
gfCNCPoint3[18380] = {X 303.3281, Y 52.9755, Z -4.6667, A 0.000, B 0.000, C 0.000 }
gfCNCPoint3[18381] = {X 304.1247, Y 52.2551, Z -4.6667, A 0.000, B 0.000, C 0.000 }
gfCNCPoint3[18382] = {X 305.0187, Y 51.6597, Z -4.6667, A 0.000, B 0.000, C 0.000 }
gfCNCPoint3[18383] = {X 306.1514, Y 51.1428, Z -4.6667, A 0.000, B 0.000, C 0.000 }
gfCNCPoint3[18384] = {X 307.3557, Y 50.8265, Z -4.6667, A 0.000, B 0.000, C 0.000 }
gfCNCPoint3[18385] = {X 308.5962, Y 50.7200, Z -4.6667, A 0.000, B 0.000, C 0.000 }
gfCNCPoint3[18386] = {X 324.3107, Y 50.7200, Z -4.6667, A 0.000, B 0.000, C 0.000 }
gfCNCPoint3[18387] = {X 325.2469, Y 50.7804, Z -4.6667, A 0.000, B 0.000, C 0.000 }
gfCNCPoint3[18388] = {X 326.1675, Y 50.9608, Z -4.6667, A 0.000, B 0.000, C 0.000 }
gfCNCPoint3[18389] = {X 326.5260, Y 51.0653, Z -4.6667, A 0.000, B 0.000, C 0.000 }
gfCNCPoint3[18390] = {X 326.8787, Y 51.1880, Z -4.6667, A 0.000, B 0.000, C 0.000 }
gfCNCPoint3[18391] = {X 327.4502, Y 51.4318, Z -4.6667, A 0.000, B 0.000, C 0.000 }
gfCNCPoint3[18392] = {X 327.9989, Y 51.7234, Z -4.6667, A 0.000, B 0.000, C 0.000 }
gfCNCPoint3[18393] = {X 328.5424, Y 52.0762, Z -4.6667, A 0.000, B 0.000, C 0.000 }
gfCNCPoint3[18394] = {X 329.0524, Y 52.4760, Z -4.6667, A 0.000, B 0.000, C 0.000 }
gfCNCPoint3[18395] = {X 329.9292, Y 53.3707, Z -4.6667, A 0.000, B 0.000, C 0.000 }
gfCNCPoint3[18396] = {X 330.6397, Y 54.4025, Z -4.6667, A 0.000, B 0.000, C 0.000 }
gfCNCPoint3[18397] = {X 331.1627, Y 55.5408, Z -4.6667, A 0.000, B 0.000, C 0.000 }
gfCNCPoint3[18398] = {X 331.4829, Y 56.7519, Z -4.6667, A 0.000, B 0.000, C 0.000 }
gfCNCPoint3[18399] = {X 331.5907, Y 58.0000, Z -4.6667, A 0.000, B 0.000, C 0.000 }
gfCNCPoint3[18400] = {X 331.5907, Y 58.9397, Z -4.6667, A 0.000, B 0.000, C 0.000 }
gfCNCPoint3[18401] = {X 331.4733, Y 60.2167, Z -4.6667, A 0.000, B 0.000, C 0.000 }
gfCNCPoint3[18402] = {X 331.1349, Y 61.4536, Z -4.6667, A 0.000, B 0.000, C 0.000 }
gfCNCPoint3[18403] = {X 330.5857, Y 62.6124, Z -4.6667, A 0.000, B 0.000, C 0.000 }
gfCNCPoint3[18404] = {X 329.8427, Y 63.6576, Z -4.6667, A 0.000, B 0.000, C 0.000 }
gfCNCPoint3[18405] = {X 328.9287, Y 64.5570, Z -4.6667, A 0.000, B 0.000, C 0.000 }
gfCNCPoint3[18406] = {X 327.8717, Y 65.2831, Z -4.6667, A 0.000, B 0.000, C 0.000 }
gfCNCPoint3[18407] = {X 327.8732, Y 83.2150, Z -4.6667, A 0.000, B 0.000, C 0.000 }
gfCNCPoint3[18408] = {X 327.8867, Y 84.5918, Z -4.6667, A 0.000, B 0.000, C 0.000 }
gfCNCPoint3[18409] = {X 327.8962, Y 84.9541, Z -4.6667, A 0.000, B 0.000, C 0.000 }
gfCNCPoint3[18410] = {X 327.9230, Y 85.3157, Z -4.6667, A 0.000, B 0.000, C 0.000 }
gfCNCPoint3[18411] = {X 328.8644, Y 85.6729, Z -4.6667, A 0.000, B 0.000, C 0.000 }
gfCNCPoint3[18412] = {X 329.8339, Y 85.9445, Z -4.6667, A 0.000, B 0.000, C 0.000 }
gfCNCPoint3[18413] = {X 332.7051, Y 86.5198, Z -4.6667, A 0.000, B 0.000, C 0.000 }
gfCNCPoint3[18414] = {X 335.6102, Y 86.8868, Z -4.6667, A 0.000, B 0.000, C 0.000 }
gfCNCPoint3[18415] = {X 339.6590, Y 87.2001, Z -4.6667, A 0.000, B 0.000, C 0.000 }
gfCNCPoint3[18416] = {X 343.7161, Y 87.3757, Z -4.6667, A 0.000, B 0.000, C 0.000 }
gfCNCPoint3[18417] = {X 347.7768, Y 87.4133, Z -4.6667, A 0.000, B 0.000, C 0.000 }
gfCNCPoint3[18418] = {X 352.0644, Y 87.3766, Z -4.6667, A 0.000, B 0.000, C 0.000 }
gfCNCPoint3[18419] = {X 356.3478, Y 87.1854, Z -4.6667, A 0.000, B 0.000, C 0.000 }
gfCNCPoint3[18420] = {X 360.6216, Y 86.8398, Z -4.6667, A 0.000, B 0.000, C 0.000 }
gfCNCPoint3[18421] = {X 362.7646, Y 86.5737, Z -4.6667, A 0.000, B 0.000, C 0.000 }
gfCNCPoint3[18422] = {X 364.8876, Y 86.1789, Z -4.6667, A 0.000, B 0.000, C 0.000 }
gfCNCPoint3[18423] = {X 366.9831, Y 85.6569, Z -4.6667, A 0.000, B 0.000, C 0.000 }
gfCNCPoint3[18424] = {X 367.4428, Y 85.5106, Z -4.6667, A 0.000, B 0.000, C 0.000 }
gfCNCPoint3[18425] = {X 367.8889, Y 85.3266, Z -4.6667, A 0.000, B 0.000, C 0.000 }
gfCNCPoint3[18426] = {X 367.9423, Y 84.5784, Z -4.6667, A 0.000, B 0.000, C 0.000 }
gfCNCPoint3[18427] = {X 367.9601, Y 83.8285, Z -4.6667, A 0.000, B 0.000, C 0.000 }
gfCNCPoint3[18428] = {X 367.9588, Y 65.2840, Z -4.6667, A 0.000, B 0.000, C 0.000 }
gfCNCPoint3[18429] = {X 366.9049, Y 64.5649, Z -4.6667, A 0.000, B 0.000, C 0.000 }
gfCNCPoint3[18430] = {X 365.9928, Y 63.6729, Z -4.6667, A 0.000, B 0.000, C 0.000 }
gfCNCPoint3[18431] = {X 365.2504, Y 62.6353, Z -4.6667, A 0.000, B 0.000, C 0.000 }
gfCNCPoint3[18432] = {X 364.7005, Y 61.4841, Z -4.6667, A 0.000, B 0.000, C 0.000 }
gfCNCPoint3[18433] = {X 364.3600, Y 60.2546, Z -4.6667, A 0.000, B 0.000, C 0.000 }
gfCNCPoint3[18434] = {X 364.2395, Y 58.9845, Z -4.6667, A 0.000, B 0.000, C 0.000 }
gfCNCPoint3[18435] = {X 364.2393, Y 58.0000, Z -4.6667, A 0.000, B 0.000, C 0.000 }
gfCNCPoint3[18436] = {X 364.3499, Y 56.7358, Z -4.6667, A 0.000, B 0.000, C 0.000 }
gfCNCPoint3[18437] = {X 364.6783, Y 55.5101, Z -4.6667, A 0.000, B 0.000, C 0.000 }
gfCNCPoint3[18438] = {X 365.2146, Y 54.3600, Z -4.6667, A 0.000, B 0.000, C 0.000 }
gfCNCPoint3[18439] = {X 365.9425, Y 53.3205, Z -4.6667, A 0.000, B 0.000, C 0.000 }
gfCNCPoint3[18440] = {X 366.8398, Y 52.4232, Z -4.6667, A 0.000, B 0.000, C 0.000 }
gfCNCPoint3[18441] = {X 367.8793, Y 51.6953, Z -4.6667, A 0.000, B 0.000, C 0.000 }
gfCNCPoint3[18442] = {X 369.0294, Y 51.1590, Z -4.6667, A 0.000, B 0.000, C 0.000 }
gfCNCPoint3[18443] = {X 370.2551, Y 50.8306, Z -4.6667, A 0.000, B 0.000, C 0.000 }
gfCNCPoint3[18444] = {X 371.5193, Y 50.7200, Z -4.6667, A 0.000, B 0.000, C 0.000 }
gfCNCPoint3[18445] = {X 388.0597, Y 50.7200, Z -4.6667, A 0.000, B 0.000, C 0.000 }
gfCNCPoint3[18446] = {X 389.2271, Y 50.8142, Z -4.6667, A 0.000, B 0.000, C 0.000 }
gfCNCPoint3[18447] = {X 390.3643, Y 51.0944, Z -4.6667, A 0.000, B 0.000, C 0.000 }
gfCNCPoint3[18448] = {X 391.4418, Y 51.5533, Z -4.6667, A 0.000, B 0.000, C 0.000 }
gfCNCPoint3[18449] = {X 392.4319, Y 52.1791, Z -4.6667, A 0.000, B 0.000, C 0.000 }
gfCNCPoint3[18450] = {X 393.3087, Y 52.9556, Z -4.6667, A 0.000, B 0.000, C 0.000 }
gfCNCPoint3[18451] = {X 394.1855, Y 52.1791, Z -4.6667, A 0.000, B 0.000, C 0.000 }
gfCNCPoint3[18452] = {X 395.1756, Y 51.5533, Z -4.6667, A 0.000, B 0.000, C 0.000 }
gfCNCPoint3[18453] = {X 396.2531, Y 51.0944, Z -4.6667, A 0.000, B 0.000, C 0.000 }
gfCNCPoint3[18454] = {X 397.3903, Y 50.8142, Z -4.6667, A 0.000, B 0.000, C 0.000 }
gfCNCPoint3[18455] = {X 398.5577, Y 50.7200, Z -4.6667, A 0.000, B 0.000, C 0.000 }
gfCNCPoint3[18456] = {X 419.4886, Y 50.7200, Z -4.6667, A 0.000, B 0.000, C 0.000 }
gfCNCPoint3[18457] = {X 420.6740, Y 50.8172, Z -4.6667, A 0.000, B 0.000, C 0.000 }
gfCNCPoint3[18458] = {X 421.8277, Y 51.1060, Z -4.6667, A 0.000, B 0.000, C 0.000 }
gfCNCPoint3[18459] = {X 422.9190, Y 51.5789, Z -4.6667, A 0.000, B 0.000, C 0.000 }
gfCNCPoint3[18460] = {X 423.9187, Y 52.2231, Z -4.6667, A 0.000, B 0.000, C 0.000 }
gfCNCPoint3[18461] = {X 424.8002, Y 53.0215, Z -4.6667, A 0.000, B 0.000, C 0.000 }
gfCNCPoint3[18462] = {X 425.5399, Y 53.9528, Z -4.6667, A 0.000, B 0.000, C 0.000 }
gfCNCPoint3[18463] = {X 426.1182, Y 54.9921, Z -4.6667, A 0.000, B 0.000, C 0.000 }
gfCNCPoint3[18464] = {X 426.5194, Y 56.1117, Z -4.6667, A 0.000, B 0.000, C 0.000 }
gfCNCPoint3[18465] = {X 430.7007, Y 57.7410, Z -4.6667, A 0.000, B 0.000, C 0.000 }
gfCNCPoint3[18466] = {X 454.8988, Y 67.3418, Z -4.6667, A 0.000, B 0.000, C 0.000 }
gfCNCPoint3[18467] = {X 454.8989, Y 65.2839, Z -4.6667, A 0.000, B 0.000, C 0.000 }
gfCNCPoint3[18468] = {X 453.8917, Y 64.6026, Z -4.6667, A 0.000, B 0.000, C 0.000 }
gfCNCPoint3[18469] = {X 453.0118, Y 63.7632, Z -4.6667, A 0.000, B 0.000, C 0.000 }
gfCNCPoint3[18470] = {X 452.2840, Y 62.7890, Z -4.6667, A 0.000, B 0.000, C 0.000 }
gfCNCPoint3[18471] = {X 451.7285, Y 61.7073, Z -4.6667, A 0.000, B 0.000, C 0.000 }
gfCNCPoint3[18472] = {X 451.4296, Y 60.8257, Z -4.6667, A 0.000, B 0.000, C 0.000 }
gfCNCPoint3[18473] = {X 451.2457, Y 59.9131, Z -4.6667, A 0.000, B 0.000, C 0.000 }
gfCNCPoint3[18474] = {X 451.1798, Y 58.9845, Z -4.6667, A 0.000, B 0.000, C 0.000 }
gfCNCPoint3[18475] = {X 451.1796, Y 58.0000, Z -4.6667, A 0.000, B 0.000, C 0.000 }
gfCNCPoint3[18476] = {X 451.2795, Y 56.7981, Z -4.6667, A 0.000, B 0.000, C 0.000 }
gfCNCPoint3[18477] = {X 451.5765, Y 55.6291, Z -4.6667, A 0.000, B 0.000, C 0.000 }
gfCNCPoint3[18478] = {X 452.0624, Y 54.5253, Z -4.6667, A 0.000, B 0.000, C 0.000 }
gfCNCPoint3[18479] = {X 452.7238, Y 53.5168, Z -4.6667, A 0.000, B 0.000, C 0.000 }
gfCNCPoint3[18480] = {X 453.5427, Y 52.6313, Z -4.6667, A 0.000, B 0.000, C 0.000 }
gfCNCPoint3[18481] = {X 454.4966, Y 51.8932, Z -4.6667, A 0.000, B 0.000, C 0.000 }
gfCNCPoint3[18482] = {X 455.4133, Y 51.3880, Z -4.6667, A 0.000, B 0.000, C 0.000 }
gfCNCPoint3[18483] = {X 456.3931, Y 51.0195, Z -4.6667, A 0.000, B 0.000, C 0.000 }
gfCNCPoint3[18484] = {X 457.4155, Y 50.7953, Z -4.6667, A 0.000, B 0.000, C 0.000 }
gfCNCPoint3[18485] = {X 458.4596, Y 50.7200, Z -4.6667, A 0.000, B 0.000, C 0.000 }
gfCNCPoint3[18486] = {X 475.0000, Y 50.7200, Z -4.6667, A 0.000, B 0.000, C 0.000 }
gfCNCPoint3[18487] = {X 476.0441, Y 50.7953, Z -4.6667, A 0.000, B 0.000, C 0.000 }
gfCNCPoint3[18488] = {X 477.0665, Y 51.0195, Z -4.6667, A 0.000, B 0.000, C 0.000 }
gfCNCPoint3[18489] = {X 478.0463, Y 51.3880, Z -4.6667, A 0.000, B 0.000, C 0.000 }
gfCNCPoint3[18490] = {X 478.9630, Y 51.8932, Z -4.6667, A 0.000, B 0.000, C 0.000 }
gfCNCPoint3[18491] = {X 479.9169, Y 52.6313, Z -4.6667, A 0.000, B 0.000, C 0.000 }
gfCNCPoint3[18492] = {X 480.7358, Y 53.5168, Z -4.6667, A 0.000, B 0.000, C 0.000 }
gfCNCPoint3[18493] = {X 481.3972, Y 54.5253, Z -4.6667, A 0.000, B 0.000, C 0.000 }
gfCNCPoint3[18494] = {X 481.8831, Y 55.6291, Z -4.6667, A 0.000, B 0.000, C 0.000 }
gfCNCPoint3[18495] = {X 482.1801, Y 56.7981, Z -4.6667, A 0.000, B 0.000, C 0.000 }
gfCNCPoint3[18496] = {X 482.2800, Y 58.0000, Z -4.6667, A 0.000, B 0.000, C 0.000 }
gfCNCPoint3[18497] = {X 482.2798, Y 58.9942, Z -4.6667, A 0.000, B 0.000, C 0.000 }
gfCNCPoint3[18498] = {X 482.1578, Y 60.2626, Z -4.6667, A 0.000, B 0.000, C 0.000 }
gfCNCPoint3[18499] = {X 481.8165, Y 61.4903, Z -4.6667, A 0.000, B 0.000, C 0.000 }
gfCNCPoint3[18500] = {X 481.2663, Y 62.6396, Z -4.6667, A 0.000, B 0.000, C 0.000 }
gfCNCPoint3[18501] = {X 480.5243, Y 63.6755, Z -4.6667, A 0.000, B 0.000, C 0.000 }
gfCNCPoint3[18502] = {X 479.6129, Y 64.5661, Z -4.6667, A 0.000, B 0.000, C 0.000 }
gfCNCPoint3[18503] = {X 478.5603, Y 65.2841, Z -4.6667, A 0.000, B 0.000, C 0.000 }
gfCNCPoint3[18504] = {X 478.5606, Y 90.7243, Z -4.6667, A 0.000, B 0.000, C 0.000 }
gfCNCPoint3[18505] = {X 479.5432, Y 91.3829, Z -4.6667, A 0.000, B 0.000, C 0.000 }
gfCNCPoint3[18506] = {X 480.4057, Y 92.1925, Z -4.6667, A 0.000, B 0.000, C 0.000 }
gfCNCPoint3[18507] = {X 481.1251, Y 93.1314, Z -4.6667, A 0.000, B 0.000, C 0.000 }
gfCNCPoint3[18508] = {X 481.6823, Y 94.1749, Z -4.6667, A 0.000, B 0.000, C 0.000 }
gfCNCPoint3[18509] = {X 482.0624, Y 95.2950, Z -4.6667, A 0.000, B 0.000, C 0.000 }
gfCNCPoint3[18510] = {X 507.6815, Y 95.2950, Z -4.6667, A 0.000, B 0.000, C 0.000 }
gfCNCPoint3[18511] = {X 507.6815, Y 97.6950, Z -4.6667, A 0.000, B 0.000, C 0.000 }
gfCNCPoint3[18512] = {X 597.6966, Y 97.6950, Z -4.6667, A 0.000, B 0.000, C 0.000 }
gfCNCPoint3[18513] = {X 597.6966, Y 51.8000, Z -4.6667, A 0.000, B 0.000, C 0.000 }
gfCNCPoint3[18514] = {X 593.5565, Y 51.8000, Z -4.6667, A 0.000, B 0.000, C 0.000 }
gfCNCPoint3[18515] = {X 592.3428, Y 51.6908, Z -4.6667, A 0.000, B 0.000, C 0.000 }
gfCNCPoint3[18516] = {X 591.1680, Y 51.3667, Z -4.6667, A 0.000, B 0.000, C 0.000 }
gfCNCPoint3[18517] = {X 590.0699, Y 50.8381, Z -4.6667, A 0.000, B 0.000, C 0.000 }
gfCNCPoint3[18518] = {X 589.0838, Y 50.1220, Z -4.6667, A 0.000, B 0.000, C 0.000 }
gfCNCPoint3[18519] = {X 588.4736, Y 49.5171, Z -4.6667, A 0.000, B 0.000, C 0.000 }
gfCNCPoint3[18520] = {X 587.9446, Y 48.8401, Z -4.6667, A 0.000, B 0.000, C 0.000 }
gfCNCPoint3[18521] = {X 587.5052, Y 48.1018, Z -4.6667, A 0.000, B 0.000, C 0.000 }
gfCNCPoint3[18522] = {X 587.0658, Y 48.8401, Z -4.6667, A 0.000, B 0.000, C 0.000 }
gfCNCPoint3[18523] = {X 586.5368, Y 49.5171, Z -4.6667, A 0.000, B 0.000, C 0.000 }
gfCNCPoint3[18524] = {X 585.9266, Y 50.1220, Z -4.6667, A 0.000, B 0.000, C 0.000 }
gfCNCPoint3[18525] = {X 585.1803, Y 50.6880, Z -4.6667, A 0.000, B 0.000, C 0.000 }
gfCNCPoint3[18526] = {X 584.3634, Y 51.1461, Z -4.6667, A 0.000, B 0.000, C 0.000 }
gfCNCPoint3[18527] = {X 583.3013, Y 51.5442, Z -4.6667, A 0.000, B 0.000, C 0.000 }
gfCNCPoint3[18528] = {X 582.1877, Y 51.7603, Z -4.6667, A 0.000, B 0.000, C 0.000 }
gfCNCPoint3[18529] = {X 581.0538, Y 51.7882, Z -4.6667, A 0.000, B 0.000, C 0.000 }
gfCNCPoint3[18530] = {X 579.9310, Y 51.6273, Z -4.6667, A 0.000, B 0.000, C 0.000 }
gfCNCPoint3[18531] = {X 578.8505, Y 51.2819, Z -4.6667, A 0.000, B 0.000, C 0.000 }
gfCNCPoint3[18532] = {X 577.8425, Y 50.7618, Z -4.6667, A 0.000, B 0.000, C 0.000 }
gfCNCPoint3[18533] = {X 576.9350, Y 50.0813, Z -4.6667, A 0.000, B 0.000, C 0.000 }
gfCNCPoint3[18534] = {X 576.3133, Y 49.4513, Z -4.6667, A 0.000, B 0.000, C 0.000 }
gfCNCPoint3[18535] = {X 575.7786, Y 48.7459, Z -4.6667, A 0.000, B 0.000, C 0.000 }
gfCNCPoint3[18536] = {X 575.3401, Y 47.9770, Z -4.6667, A 0.000, B 0.000, C 0.000 }
gfCNCPoint3[18537] = {X 574.9017, Y 48.7459, Z -4.6667, A 0.000, B 0.000, C 0.000 }
gfCNCPoint3[18538] = {X 574.3670, Y 49.4513, Z -4.6667, A 0.000, B 0.000, C 0.000 }
gfCNCPoint3[18539] = {X 573.7453, Y 50.0813, Z -4.6667, A 0.000, B 0.000, C 0.000 }
gfCNCPoint3[18540] = {X 572.7526, Y 50.8143, Z -4.6667, A 0.000, B 0.000, C 0.000 }
gfCNCPoint3[18541] = {X 571.6437, Y 51.3558, Z -4.6667, A 0.000, B 0.000, C 0.000 }
gfCNCPoint3[18542] = {X 570.4553, Y 51.6880, Z -4.6667, A 0.000, B 0.000, C 0.000 }
gfCNCPoint3[18543] = {X 569.2264, Y 51.8000, Z -4.6667, A 0.000, B 0.000, C 0.000 }
gfCNCPoint3[18544] = {X 562.4443, Y 51.8000, Z -4.6667, A 0.000, B 0.000, C 0.000 }
gfCNCPoint3[18545] = {X 561.2635, Y 51.6967, Z -4.6667, A 0.000, B 0.000, C 0.000 }
gfCNCPoint3[18546] = {X 560.1186, Y 51.3899, Z -4.6667, A 0.000, B 0.000, C 0.000 }
gfCNCPoint3[18547] = {X 559.0443, Y 50.8890, Z -4.6667, A 0.000, B 0.000, C 0.000 }
gfCNCPoint3[18548] = {X 558.0733, Y 50.2091, Z -4.6667, A 0.000, B 0.000, C 0.000 }
gfCNCPoint3[18549] = {X 557.2352, Y 49.3710, Z -4.6667, A 0.000, B 0.000, C 0.000 }
gfCNCPoint3[18550] = {X 556.5553, Y 48.4000, Z -4.6667, A 0.000, B 0.000, C 0.000 }
gfCNCPoint3[18551] = {X 556.0544, Y 47.3257, Z -4.6667, A 0.000, B 0.000, C 0.000 }
gfCNCPoint3[18552] = {X 555.7476, Y 46.1808, Z -4.6667, A 0.000, B 0.000, C 0.000 }
gfCNCPoint3[18553] = {X 555.6443, Y 45.0000, Z -4.6667, A 0.000, B 0.000, C 0.000 }
gfCNCPoint3[18554] = {X 555.6443, Y 44.0544, Z -4.6667, A 0.000, B 0.000, C 0.000 }
gfCNCPoint3[18555] = {X 555.7469, Y 42.9027, Z -4.6667, A 0.000, B 0.000, C 0.000 }
gfCNCPoint3[18556] = {X 556.0422, Y 41.7847, Z -4.6667, A 0.000, B 0.000, C 0.000 }
gfCNCPoint3[18557] = {X 556.5217, Y 40.7326, Z -4.6667, A 0.000, B 0.000, C 0.000 }
gfCNCPoint3[18558] = {X 557.1718, Y 39.7763, Z -4.6667, A 0.000, B 0.000, C 0.000 }
gfCNCPoint3[18559] = {X 557.1718, Y 10.2283, Z -4.6667, A 0.000, B 0.000, C 0.000 }
gfCNCPoint3[18560] = {X 556.5257, Y 9.2823, Z -4.6667, A 0.000, B 0.000, C 0.000 }
gfCNCPoint3[18561] = {X 556.0477, Y 8.2413, Z -4.6667, A 0.000, B 0.000, C 0.000 }
gfCNCPoint3[18562] = {X 555.7511, Y 7.1347, Z -4.6667, A 0.000, B 0.000, C 0.000 }
gfCNCPoint3[18563] = {X 555.6446, Y 5.9941, Z -4.6667, A 0.000, B 0.000, C 0.000 }
gfCNCPoint3[18564] = {X 555.6443, Y 5.0000, Z -4.6667, A 0.000, B 0.000, C 0.000 }
gfCNCPoint3[18565] = {X 555.6452, Y 4.8910, Z -4.6667, A 0.000, B 0.000, C 0.000 }
gfCNCPoint3[18566] = {X 555.6478, Y 4.7819, Z -4.6667, A 0.000, B 0.000, C 0.000 }
gfCNCPoint3[18567] = {X 555.8079, Y 3.5174, Z -4.6667, A 0.000, B 0.000, C 0.000 }
gfCNCPoint3[18568] = {X 556.2012, Y 2.3050, Z -4.6667, A 0.000, B 0.000, C 0.000 }
gfCNCPoint3[18569] = {X 358.2593, Y 2.3050, Z -4.6667, A 0.000, B 0.000, C 0.000 }
gfCNCPoint3[18570] = {X 360.1206, Y 3.4746, Z -4.6667, A 0.000, B 0.000, C 0.000 }
gfCNCPoint3[18571] = {X 361.8533, Y 4.8275, Z -4.6667, A 0.000, B 0.000, C 0.000 }
gfCNCPoint3[18572] = {X 363.4393, Y 6.3496, Z -4.6667, A 0.000, B 0.000, C 0.000 }
gfCNCPoint3[18573] = {X 363.7857, Y 6.7266, Z -4.6667, A 0.000, B 0.000, C 0.000 }
gfCNCPoint3[18574] = {X 364.1230, Y 7.1116, Z -4.6667, A 0.000, B 0.000, C 0.000 }
gfCNCPoint3[18575] = {X 365.6206, Y 9.0444, Z -4.6667, A 0.000, B 0.000, C 0.000 }
gfCNCPoint3[18576] = {X 366.9245, Y 11.1130, Z -4.6667, A 0.000, B 0.000, C 0.000 }
gfCNCPoint3[18577] = {X 368.0224, Y 13.2978, Z -4.6667, A 0.000, B 0.000, C 0.000 }
gfCNCPoint3[18578] = {X 368.9041, Y 15.5785, Z -4.6667, A 0.000, B 0.000, C 0.000 }
gfCNCPoint3[18579] = {X 369.5613, Y 17.9337, Z -4.6667, A 0.000, B 0.000, C 0.000 }
gfCNCPoint3[18580] = {X 370.0535, Y 20.6185, Z -4.6667, A 0.000, B 0.000, C 0.000 }
gfCNCPoint3[18581] = {X 370.3162, Y 23.3354, Z -4.6667, A 0.000, B 0.000, C 0.000 }
gfCNCPoint3[18582] = {X 370.3478, Y 26.0648, Z -4.6667, A 0.000, B 0.000, C 0.000 }
gfCNCPoint3[18583] = {X 370.1478, Y 28.7870, Z -4.6667, A 0.000, B 0.000, C 0.000 }
gfCNCPoint3[18584] = {X 369.7178, Y 31.4825, Z -4.6667, A 0.000, B 0.000, C 0.000 }
gfCNCPoint3[18585] = {X 369.1821, Y 33.6341, Z -4.6667, A 0.000, B 0.000, C 0.000 }
gfCNCPoint3[18586] = {X 368.4585, Y 35.7300, Z -4.6667, A 0.000, B 0.000, C 0.000 }
gfCNCPoint3[18587] = {X 367.5526, Y 37.7539, Z -4.6667, A 0.000, B 0.000, C 0.000 }
gfCNCPoint3[18588] = {X 366.4715, Y 39.6898, Z -4.6667, A 0.000, B 0.000, C 0.000 }
gfCNCPoint3[18589] = {X 365.2237, Y 41.5227, Z -4.6667, A 0.000, B 0.000, C 0.000 }
gfCNCPoint3[18590] = {X 365.0834, Y 41.7130, Z -4.6667, A 0.000, B 0.000, C 0.000 }
gfCNCPoint3[18591] = {X 364.4589, Y 42.4798, Z -4.6667, A 0.000, B 0.000, C 0.000 }
gfCNCPoint3[18592] = {X 363.1646, Y 43.9320, Z -4.6667, A 0.000, B 0.000, C 0.000 }
gfCNCPoint3[18593] = {X 361.7464, Y 45.2634, Z -4.6667, A 0.000, B 0.000, C 0.000 }
gfCNCPoint3[18594] = {X 360.2154, Y 46.4634, Z -4.6667, A 0.000, B 0.000, C 0.000 }
gfCNCPoint3[18595] = {X 358.5837, Y 47.5226, Z -4.6667, A 0.000, B 0.000, C 0.000 }
gfCNCPoint3[18596] = {X 356.8644, Y 48.4325, Z -4.6667, A 0.000, B 0.000, C 0.000 }
gfCNCPoint3[18597] = {X 356.4678, Y 48.6203, Z -4.6667, A 0.000, B 0.000, C 0.000 }
gfCNCPoint3[18598] = {X 354.6708, Y 49.3142, Z -4.6667, A 0.000, B 0.000, C 0.000 }
gfCNCPoint3[18599] = {X 352.8232, Y 49.8592, Z -4.6667, A 0.000, B 0.000, C 0.000 }
gfCNCPoint3[18600] = {X 350.9372, Y 50.2515, Z -4.6667, A 0.000, B 0.000, C 0.000 }
gfCNCPoint3[18601] = {X 349.0255, Y 50.4886, Z -4.6667, A 0.000, B 0.000, C 0.000 }
gfCNCPoint3[18602] = {X 347.1008, Y 50.5689, Z -4.6667, A 0.000, B 0.000, C 0.000 }
gfCNCPoint3[18603] = {X 344.9874, Y 50.5327, Z -4.6667, A 0.000, B 0.000, C 0.000 }
gfCNCPoint3[18604] = {X 342.8850, Y 50.3135, Z -4.6667, A 0.000, B 0.000, C 0.000 }
gfCNCPoint3[18605] = {X 340.8096, Y 49.9130, Z -4.6667, A 0.000, B 0.000, C 0.000 }
gfCNCPoint3[18606] = {X 338.7767, Y 49.3340, Z -4.6667, A 0.000, B 0.000, C 0.000 }
gfCNCPoint3[18607] = {X 336.8016, Y 48.5811, Z -4.6667, A 0.000, B 0.000, C 0.000 }
gfCNCPoint3[18608] = {X 334.8991, Y 47.6598, Z -4.6667, A 0.000, B 0.000, C 0.000 }
gfCNCPoint3[18609] = {X 333.3418, Y 46.7036, Z -4.6667, A 0.000, B 0.000, C 0.000 }
gfCNCPoint3[18610] = {X 331.8605, Y 45.6333, Z -4.6667, A 0.000, B 0.000, C 0.000 }
gfCNCPoint3[18611] = {X 330.4637, Y 44.4550, Z -4.6667, A 0.000, B 0.000, C 0.000 }
gfCNCPoint3[18612] = {X 329.4664, Y 44.4078, Z -4.6667, A 0.000, B 0.000, C 0.000 }
gfCNCPoint3[18613] = {X 328.4996, Y 44.1587, Z -4.6667, A 0.000, B 0.000, C 0.000 }
gfCNCPoint3[18614] = {X 327.6038, Y 43.7181, Z -4.6667, A 0.000, B 0.000, C 0.000 }
gfCNCPoint3[18615] = {X 326.8164, Y 43.1044, Z -4.6667, A 0.000, B 0.000, C 0.000 }
gfCNCPoint3[18616] = {X 326.1897, Y 42.4934, Z -4.6667, A 0.000, B 0.000, C 0.000 }
gfCNCPoint3[18617] = {X 325.5686, Y 41.7541, Z -4.6667, A 0.000, B 0.000, C 0.000 }
gfCNCPoint3[18618] = {X 325.1052, Y 40.9070, Z -4.6667, A 0.000, B 0.000, C 0.000 }
gfCNCPoint3[18619] = {X 324.8177, Y 39.9852, Z -4.6667, A 0.000, B 0.000, C 0.000 }
gfCNCPoint3[18620] = {X 324.7172, Y 39.0249, Z -4.6667, A 0.000, B 0.000, C 0.000 }
gfCNCPoint3[18621] = {X 324.8079, Y 38.0635, Z -4.6667, A 0.000, B 0.000, C 0.000 }
gfCNCPoint3[18622] = {X 325.0860, Y 37.1389, Z -4.6667, A 0.000, B 0.000, C 0.000 }
gfCNCPoint3[18623] = {X 325.5408, Y 36.2871, Z -4.6667, A 0.000, B 0.000, C 0.000 }
gfCNCPoint3[18624] = {X 329.7765, Y 29.9538, Z -4.6667, A 0.000, B 0.000, C 0.000 }
gfCNCPoint3[18625] = {X 330.4614, Y 29.1399, Z -4.6667, A 0.000, B 0.000, C 0.000 }
gfCNCPoint3[18626] = {X 331.3063, Y 28.4938, Z -4.6667, A 0.000, B 0.000, C 0.000 }
gfCNCPoint3[18627] = {X 332.2711, Y 28.0462, Z -4.6667, A 0.000, B 0.000, C 0.000 }
gfCNCPoint3[18628] = {X 333.3101, Y 27.8182, Z -4.6667, A 0.000, B 0.000, C 0.000 }
gfCNCPoint3[18629] = {X 334.3737, Y 27.8207, Z -4.6667, A 0.000, B 0.000, C 0.000 }
gfCNCPoint3[18630] = {X 335.4116, Y 28.0536, Z -4.6667, A 0.000, B 0.000, C 0.000 }
gfCNCPoint3[18631] = {X 336.3743, Y 28.5058, Z -4.6667, A 0.000, B 0.000, C 0.000 }
gfCNCPoint3[18632] = {X 337.2162, Y 29.1559, Z -4.6667, A 0.000, B 0.000, C 0.000 }
gfCNCPoint3[18633] = {X 337.7895, Y 29.7082, Z -4.6667, A 0.000, B 0.000, C 0.000 }
gfCNCPoint3[18634] = {X 338.3584, Y 30.3646, Z -4.6667, A 0.000, B 0.000, C 0.000 }
gfCNCPoint3[18635] = {X 338.8019, Y 31.1116, Z -4.6667, A 0.000, B 0.000, C 0.000 }
gfCNCPoint3[18636] = {X 339.1060, Y 31.9253, Z -4.6667, A 0.000, B 0.000, C 0.000 }
gfCNCPoint3[18637] = {X 339.2610, Y 32.7801, Z -4.6667, A 0.000, B 0.000, C 0.000 }
gfCNCPoint3[18638] = {X 339.2619, Y 33.6488, Z -4.6667, A 0.000, B 0.000, C 0.000 }
gfCNCPoint3[18639] = {X 339.9076, Y 34.2206, Z -4.6667, A 0.000, B 0.000, C 0.000 }
gfCNCPoint3[18640] = {X 340.5765, Y 34.7651, Z -4.6667, A 0.000, B 0.000, C 0.000 }
gfCNCPoint3[18641] = {X 341.8083, Y 35.5731, Z -4.6667, A 0.000, B 0.000, C 0.000 }
gfCNCPoint3[18642] = {X 343.1448, Y 36.1926, Z -4.6667, A 0.000, B 0.000, C 0.000 }
gfCNCPoint3[18643] = {X 344.5576, Y 36.6103, Z -4.6667, A 0.000, B 0.000, C 0.000 }
gfCNCPoint3[18644] = {X 346.0161, Y 36.8172, Z -4.6667, A 0.000, B 0.000, C 0.000 }
gfCNCPoint3[18645] = {X 347.4893, Y 36.8089, Z -4.6667, A 0.000, B 0.000, C 0.000 }
gfCNCPoint3[18646] = {X 348.8387, Y 36.6277, Z -4.6667, A 0.000, B 0.000, C 0.000 }
gfCNCPoint3[18647] = {X 350.1406, Y 36.2293, Z -4.6667, A 0.000, B 0.000, C 0.000 }
gfCNCPoint3[18648] = {X 351.3602, Y 35.6242, Z -4.6667, A 0.000, B 0.000, C 0.000 }
gfCNCPoint3[18649] = {X 352.4651, Y 34.8287, Z -4.6667, A 0.000, B 0.000, C 0.000 }
gfCNCPoint3[18650] = {X 353.5664, Y 33.7589, Z -4.6667, A 0.000, B 0.000, C 0.000 }
gfCNCPoint3[18651] = {X 354.5195, Y 32.5552, Z -4.6667, A 0.000, B 0.000, C 0.000 }
gfCNCPoint3[18652] = {X 355.3083, Y 31.2380, Z -4.6667, A 0.000, B 0.000, C 0.000 }
gfCNCPoint3[18653] = {X 355.9194, Y 29.8296, Z -4.6667, A 0.000, B 0.000, C 0.000 }
gfCNCPoint3[18654] = {X 356.3426, Y 28.3537, Z -4.6667, A 0.000, B 0.000, C 0.000 }
gfCNCPoint3[18655] = {X 356.6071, Y 26.7186, Z -4.6667, A 0.000, B 0.000, C 0.000 }
gfCNCPoint3[18656] = {X 356.7148, Y 25.0657, Z -4.6667, A 0.000, B 0.000, C 0.000 }
gfCNCPoint3[18657] = {X 356.6647, Y 23.4100, Z -4.6667, A 0.000, B 0.000, C 0.000 }
gfCNCPoint3[18658] = {X 356.4573, Y 21.7667, Z -4.6667, A 0.000, B 0.000, C 0.000 }
gfCNCPoint3[18659] = {X 356.1204, Y 20.3208, Z -4.6667, A 0.000, B 0.000, C 0.000 }
gfCNCPoint3[18660] = {X 355.5966, Y 18.9317, Z -4.6667, A 0.000, B 0.000, C 0.000 }
gfCNCPoint3[18661] = {X 354.8949, Y 17.6235, Z -4.6667, A 0.000, B 0.000, C 0.000 }
gfCNCPoint3[18662] = {X 354.0275, Y 16.4187, Z -4.6667, A 0.000, B 0.000, C 0.000 }
gfCNCPoint3[18663] = {X 353.2100, Y 15.5478, Z -4.6667, A 0.000, B 0.000, C 0.000 }
gfCNCPoint3[18664] = {X 352.2795, Y 14.7988, Z -4.6667, A 0.000, B 0.000, C 0.000 }
gfCNCPoint3[18665] = {X 351.2542, Y 14.1860, Z -4.6667, A 0.000, B 0.000, C 0.000 }
gfCNCPoint3[18666] = {X 350.1538, Y 13.7214, Z -4.6667, A 0.000, B 0.000, C 0.000 }
gfCNCPoint3[18667] = {X 348.9996, Y 13.4139, Z -4.6667, A 0.000, B 0.000, C 0.000 }
gfCNCPoint3[18668] = {X 347.3622, Y 13.2071, Z -4.6667, A 0.000, B 0.000, C 0.000 }
gfCNCPoint3[18669] = {X 345.7118, Y 13.2123, Z -4.6667, A 0.000, B 0.000, C 0.000 }
gfCNCPoint3[18670] = {X 344.0758, Y 13.4295, Z -4.6667, A 0.000, B 0.000, C 0.000 }
gfCNCPoint3[18671] = {X 342.4812, Y 13.8550, Z -4.6667, A 0.000, B 0.000, C 0.000 }
gfCNCPoint3[18672] = {X 340.9545, Y 14.4818, Z -4.6667, A 0.000, B 0.000, C 0.000 }
gfCNCPoint3[18673] = {X 339.5210, Y 15.2995, Z -4.6667, A 0.000, B 0.000, C 0.000 }
gfCNCPoint3[18674] = {X 339.4272, Y 16.1852, Z -4.6667, A 0.000, B 0.000, C 0.000 }
gfCNCPoint3[18675] = {X 339.1740, Y 17.0391, Z -4.6667, A 0.000, B 0.000, C 0.000 }
gfCNCPoint3[18676] = {X 338.7698, Y 17.8328, Z -4.6667, A 0.000, B 0.000, C 0.000 }
gfCNCPoint3[18677] = {X 338.2281, Y 18.5398, Z -4.6667, A 0.000, B 0.000, C 0.000 }
gfCNCPoint3[18678] = {X 337.5670, Y 19.1366, Z -4.6667, A 0.000, B 0.000, C 0.000 }
gfCNCPoint3[18679] = {X 336.8399, Y 19.6716, Z -4.6667, A 0.000, B 0.000, C 0.000 }
gfCNCPoint3[18680] = {X 335.9170, Y 20.1909, Z -4.6667, A 0.000, B 0.000, C 0.000 }
gfCNCPoint3[18681] = {X 334.9039, Y 20.4988, Z -4.6667, A 0.000, B 0.000, C 0.000 }
gfCNCPoint3[18682] = {X 333.8481, Y 20.5809, Z -4.6667, A 0.000, B 0.000, C 0.000 }
gfCNCPoint3[18683] = {X 332.7995, Y 20.4334, Z -4.6667, A 0.000, B 0.000, C 0.000 }
gfCNCPoint3[18684] = {X 331.8074, Y 20.0631, Z -4.6667, A 0.000, B 0.000, C 0.000 }
gfCNCPoint3[18685] = {X 330.9186, Y 19.4875, Z -4.6667, A 0.000, B 0.000, C 0.000 }
gfCNCPoint3[18686] = {X 330.1748, Y 18.7338, Z -4.6667, A 0.000, B 0.000, C 0.000 }
gfCNCPoint3[18687] = {X 329.6111, Y 17.8373, Z -4.6667, A 0.000, B 0.000, C 0.000 }
gfCNCPoint3[18688] = {X 326.0906, Y 10.5950, Z -4.6667, A 0.000, B 0.000, C 0.000 }
gfCNCPoint3[18689] = {X 325.7555, Y 9.6856, Z -4.6667, A 0.000, B 0.000, C 0.000 }
gfCNCPoint3[18690] = {X 325.6067, Y 8.7279, Z -4.6667, A 0.000, B 0.000, C 0.000 }
gfCNCPoint3[18691] = {X 325.6502, Y 7.7597, Z -4.6667, A 0.000, B 0.000, C 0.000 }
gfCNCPoint3[18692] = {X 325.8842, Y 6.8192, Z -4.6667, A 0.000, B 0.000, C 0.000 }
gfCNCPoint3[18693] = {X 326.2994, Y 5.9434, Z -4.6667, A 0.000, B 0.000, C 0.000 }
gfCNCPoint3[18694] = {X 326.9295, Y 5.1131, Z -4.6667, A 0.000, B 0.000, C 0.000 }
gfCNCPoint3[18695] = {X 327.7216, Y 4.4356, Z -4.6667, A 0.000, B 0.000, C 0.000 }
gfCNCPoint3[18696] = {X 328.3967, Y 3.9733, Z -4.6667, A 0.000, B 0.000, C 0.000 }
gfCNCPoint3[18697] = {X 329.3294, Y 3.4828, Z -4.6667, A 0.000, B 0.000, C 0.000 }
gfCNCPoint3[18698] = {X 330.3456, Y 3.2040, Z -4.6667, A 0.000, B 0.000, C 0.000 }
gfCNCPoint3[18699] = {X 331.3980, Y 3.1498, Z -4.6667, A 0.000, B 0.000, C 0.000 }
gfCNCPoint3[18700] = {X 332.4374, Y 3.3229, Z -4.6667, A 0.000, B 0.000, C 0.000 }
gfCNCPoint3[18701] = {X 333.3748, Y 2.7963, Z -4.6667, A 0.000, B 0.000, C 0.000 }
gfCNCPoint3[18702] = {X 334.3310, Y 2.3050, Z -4.6667, A 0.000, B 0.000, C 0.000 }
gfCNCPoint3[18703] = {X 334.5424, Y 2.7359, Z -4.6667, A 0.000, B 0.000, C 0.000 }
gfCNCPoint3[18704] = {X 335.0192, Y 2.5075, Z -4.6667, A 0.000, B 0.000, C 0.000 }
gfCNCPoint3[18705] = {X 335.5002, Y 2.2880, Z -4.6667, A 0.000, B 0.000, C 0.000 }
gfCNCPoint3[18706] = {X 335.8480, Y 2.1331, Z -4.6667, A 0.000, B 0.000, C 0.000 }
gfCNCPoint3[18707] = {X 337.9512, Y 1.3126, Z -4.6667, A 0.000, B 0.000, C 0.000 }
gfCNCPoint3[18708] = {X 340.1169, Y 0.6751, Z -4.6667, A 0.000, B 0.000, C 0.000 }
gfCNCPoint3[18709] = {X 342.3292, Y 0.2252, Z -4.6667, A 0.000, B 0.000, C 0.000 }
gfCNCPoint3[18710] = {X 344.5719, Y -0.0338, Z -4.6667, A 0.000, B 0.000, C 0.000 }
gfCNCPoint3[18711] = {X 346.8285, Y -0.0999, Z -4.6667, A 0.000, B 0.000, C 0.000 }
gfCNCPoint3[18712] = {X 349.0825, Y 0.0273, Z -4.6667, A 0.000, B 0.000, C 0.000 }
gfCNCPoint3[18713] = {X 351.3173, Y 0.3469, Z -4.6667, A 0.000, B 0.000, C 0.000 }
gfCNCPoint3[18714] = {X 351.8880, Y 0.4533, Z -4.6667, A 0.000, B 0.000, C 0.000 }
gfCNCPoint3[18715] = {X 353.8301, Y 0.9412, Z -4.6667, A 0.000, B 0.000, C 0.000 }
gfCNCPoint3[18716] = {X 355.7171, Y 1.6110, Z -4.6667, A 0.000, B 0.000, C 0.000 }
gfCNCPoint3[18717] = {X 357.5321, Y 2.4567, Z -4.6667, A 0.000, B 0.000, C 0.000 }
gfCNCPoint3[18718] = {X 359.2588, Y 3.4707, Z -4.6667, A 0.000, B 0.000, C 0.000 }
gfCNCPoint3[18719] = {X 360.8816, Y 4.6437, Z -4.6667, A 0.000, B 0.000, C 0.000 }
gfCNCPoint3[18720] = {X 362.3859, Y 5.9653, Z -4.6667, A 0.000, B 0.000, C 0.000 }
gfCNCPoint3[18721] = {X 363.7582, Y 7.4236, Z -4.6667, A 0.000, B 0.000, C 0.000 }
gfCNCPoint3[18722] = {X 365.2274, Y 9.3197, Z -4.6667, A 0.000, B 0.000, C 0.000 }
gfCNCPoint3[18723] = {X 366.5065, Y 11.3490, Z -4.6667, A 0.000, B 0.000, C 0.000 }
gfCNCPoint3[18724] = {X 367.5836, Y 13.4923, Z -4.6667, A 0.000, B 0.000, C 0.000 }
gfCNCPoint3[18725] = {X 368.4486, Y 15.7297, Z -4.6667, A 0.000, B 0.000, C 0.000 }
gfCNCPoint3[18726] = {X 369.0933, Y 18.0402, Z -4.6667, A 0.000, B 0.000, C 0.000 }
gfCNCPoint3[18727] = {X 369.5781, Y 20.6849, Z -4.6667, A 0.000, B 0.000, C 0.000 }
gfCNCPoint3[18728] = {X 369.8369, Y 23.3613, Z -4.6667, A 0.000, B 0.000, C 0.000 }
gfCNCPoint3[18729] = {X 369.8680, Y 26.0499, Z -4.6667, A 0.000, B 0.000, C 0.000 }
gfCNCPoint3[18730] = {X 369.6710, Y 28.7315, Z -4.6667, A 0.000, B 0.000, C 0.000 }
gfCNCPoint3[18731] = {X 369.2475, Y 31.3868, Z -4.6667, A 0.000, B 0.000, C 0.000 }
gfCNCPoint3[18732] = {X 368.7219, Y 33.4979, Z -4.6667, A 0.000, B 0.000, C 0.000 }
gfCNCPoint3[18733] = {X 368.0118, Y 35.5543, Z -4.6667, A 0.000, B 0.000, C 0.000 }
gfCNCPoint3[18734] = {X 367.1229, Y 37.5399, Z -4.6667, A 0.000, B 0.000, C 0.000 }
gfCNCPoint3[18735] = {X 366.0621, Y 39.4393, Z -4.6667, A 0.000, B 0.000, C 0.000 }
gfCNCPoint3[18736] = {X 364.8376, Y 41.2375, Z -4.6667, A 0.000, B 0.000, C 0.000 }
gfCNCPoint3[18737] = {X 364.7112, Y 41.4099, Z -4.6667, A 0.000, B 0.000, C 0.000 }
gfCNCPoint3[18738] = {X 364.0867, Y 42.1767, Z -4.6667, A 0.000, B 0.000, C 0.000 }
gfCNCPoint3[18739] = {X 362.8209, Y 43.5970, Z -4.6667, A 0.000, B 0.000, C 0.000 }
gfCNCPoint3[18740] = {X 361.4338, Y 44.8991, Z -4.6667, A 0.000, B 0.000, C 0.000 }
gfCNCPoint3[18741] = {X 359.9364, Y 46.0728, Z -4.6667, A 0.000, B 0.000, C 0.000 }
gfCNCPoint3[18742] = {X 358.3406, Y 47.1087, Z -4.6667, A 0.000, B 0.000, C 0.000 }
gfCNCPoint3[18743] = {X 356.6590, Y 47.9987, Z -4.6667, A 0.000, B 0.000, C 0.000 }
gfCNCPoint3[18744] = {X 356.2499, Y 48.1921, Z -4.6667, A 0.000, B 0.000, C 0.000 }
gfCNCPoint3[18745] = {X 354.0456, Y 49.0146, Z -4.6667, A 0.000, B 0.000, C 0.000 }
gfCNCPoint3[18746] = {X 351.7691, Y 49.6085, Z -4.6667, A 0.000, B 0.000, C 0.000 }
gfCNCPoint3[18747] = {X 349.4440, Y 49.9679, Z -4.6667, A 0.000, B 0.000, C 0.000 }
gfCNCPoint3[18748] = {X 347.0943, Y 50.0889, Z -4.6667, A 0.000, B 0.000, C 0.000 }
gfCNCPoint3[18749] = {X 345.0202, Y 50.0538, Z -4.6667, A 0.000, B 0.000, C 0.000 }
gfCNCPoint3[18750] = {X 342.9569, Y 49.8389, Z -4.6667, A 0.000, B 0.000, C 0.000 }
gfCNCPoint3[18751] = {X 340.9201, Y 49.4458, Z -4.6667, A 0.000, B 0.000, C 0.000 }
gfCNCPoint3[18752] = {X 338.9251, Y 48.8775, Z -4.6667, A 0.000, B 0.000, C 0.000 }
gfCNCPoint3[18753] = {X 336.9868, Y 48.1382, Z -4.6667, A 0.000, B 0.000, C 0.000 }
gfCNCPoint3[18754] = {X 335.1201, Y 47.2335, Z -4.6667, A 0.000, B 0.000, C 0.000 }
gfCNCPoint3[18755] = {X 333.5416, Y 46.2598, Z -4.6667, A 0.000, B 0.000, C 0.000 }
gfCNCPoint3[18756] = {X 332.0434, Y 45.1666, Z -4.6667, A 0.000, B 0.000, C 0.000 }
gfCNCPoint3[18757] = {X 330.6346, Y 43.9603, Z -4.6667, A 0.000, B 0.000, C 0.000 }
gfCNCPoint3[18758] = {X 329.6760, Y 43.9518, Z -4.6667, A 0.000, B 0.000, C 0.000 }
gfCNCPoint3[18759] = {X 328.7420, Y 43.7358, Z -4.6667, A 0.000, B 0.000, C 0.000 }
gfCNCPoint3[18760] = {X 327.8770, Y 43.3228, Z -4.6667, A 0.000, B 0.000, C 0.000 }
gfCNCPoint3[18761] = {X 327.1220, Y 42.7321, Z -4.6667, A 0.000, B 0.000, C 0.000 }
gfCNCPoint3[18762] = {X 326.5249, Y 42.1498, Z -4.6667, A 0.000, B 0.000, C 0.000 }
gfCNCPoint3[18763] = {X 325.8848, Y 41.3619, Z -4.6667, A 0.000, B 0.000, C 0.000 }
gfCNCPoint3[18764] = {X 325.4424, Y 40.4483, Z -4.6667, A 0.000, B 0.000, C 0.000 }
gfCNCPoint3[18765] = {X 325.2210, Y 39.4576, Z -4.6667, A 0.000, B 0.000, C 0.000 }
gfCNCPoint3[18766] = {X 325.2326, Y 38.4426, Z -4.6667, A 0.000, B 0.000, C 0.000 }
gfCNCPoint3[18767] = {X 325.4765, Y 37.4572, Z -4.6667, A 0.000, B 0.000, C 0.000 }
gfCNCPoint3[18768] = {X 325.9397, Y 36.5539, Z -4.6667, A 0.000, B 0.000, C 0.000 }
gfCNCPoint3[18769] = {X 330.1988, Y 30.1861, Z -4.6667, A 0.000, B 0.000, C 0.000 }
gfCNCPoint3[18770] = {X 330.8195, Y 29.4619, Z -4.6667, A 0.000, B 0.000, C 0.000 }
gfCNCPoint3[18771] = {X 331.5816, Y 28.8884, Z -4.6667, A 0.000, B 0.000, C 0.000 }
gfCNCPoint3[18772] = {X 332.4495, Y 28.4927, Z -4.6667, A 0.000, B 0.000, C 0.000 }
gfCNCPoint3[18773] = {X 333.3822, Y 28.2932, Z -4.6667, A 0.000, B 0.000, C 0.000 }
gfCNCPoint3[18774] = {X 334.3360, Y 28.2995, Z -4.6667, A 0.000, B 0.000, C 0.000 }
gfCNCPoint3[18775] = {X 335.2660, Y 28.5111, Z -4.6667, A 0.000, B 0.000, C 0.000 }
gfCNCPoint3[18776] = {X 336.1286, Y 28.9182, Z -4.6667, A 0.000, B 0.000, C 0.000 }
gfCNCPoint3[18777] = {X 336.8831, Y 29.5016, Z -4.6667, A 0.000, B 0.000, C 0.000 }
gfCNCPoint3[18778] = {X 337.4845, Y 30.0811, Z -4.6667, A 0.000, B 0.000, C 0.000 }
gfCNCPoint3[18779] = {X 338.1273, Y 30.8802, Z -4.6667, A 0.000, B 0.000, C 0.000 }
gfCNCPoint3[18780] = {X 338.5676, Y 31.8064, Z -4.6667, A 0.000, B 0.000, C 0.000 }
gfCNCPoint3[18781] = {X 338.7816, Y 32.8094, Z -4.6667, A 0.000, B 0.000, C 0.000 }
gfCNCPoint3[18782] = {X 338.7576, Y 33.8346, Z -4.6667, A 0.000, B 0.000, C 0.000 }
gfCNCPoint3[18783] = {X 339.5048, Y 34.5077, Z -4.6667, A 0.000, B 0.000, C 0.000 }
gfCNCPoint3[18784] = {X 340.2829, Y 35.1449, Z -4.6667, A 0.000, B 0.000, C 0.000 }
gfCNCPoint3[18785] = {X 341.4942, Y 35.9467, Z -4.6667, A 0.000, B 0.000, C 0.000 }
gfCNCPoint3[18786] = {X 342.8042, Y 36.5743, Z -4.6667, A 0.000, B 0.000, C 0.000 }
gfCNCPoint3[18787] = {X 344.1881, Y 37.0159, Z -4.6667, A 0.000, B 0.000, C 0.000 }
gfCNCPoint3[18788] = {X 345.6195, Y 37.2631, Z -4.6667, A 0.000, B 0.000, C 0.000 }
gfCNCPoint3[18789] = {X 347.0714, Y 37.3111, Z -4.6667, A 0.000, B 0.000, C 0.000 }
gfCNCPoint3[18790] = {X 347.5141, Y 37.2882, Z -4.6667, A 0.000, B 0.000, C 0.000 }
gfCNCPoint3[18791] = {X 348.9412, Y 37.0966, Z -4.6667, A 0.000, B 0.000, C 0.000 }
gfCNCPoint3[18792] = {X 350.3180, Y 36.6752, Z -4.6667, A 0.000, B 0.000, C 0.000 }
gfCNCPoint3[18793] = {X 351.6079, Y 36.0353, Z -4.6667, A 0.000, B 0.000, C 0.000 }
gfCNCPoint3[18794] = {X 352.7765, Y 35.1940, Z -4.6667, A 0.000, B 0.000, C 0.000 }
gfCNCPoint3[18795] = {X 353.9227, Y 34.0805, Z -4.6667, A 0.000, B 0.000, C 0.000 }
gfCNCPoint3[18796] = {X 354.9147, Y 32.8276, Z -4.6667, A 0.000, B 0.000, C 0.000 }
gfCNCPoint3[18797] = {X 355.7356, Y 31.4566, Z -4.6667, A 0.000, B 0.000, C 0.000 }
gfCNCPoint3[18798] = {X 356.3716, Y 29.9905, Z -4.6667, A 0.000, B 0.000, C 0.000 }
gfCNCPoint3[18799] = {X 356.8119, Y 28.4543, Z -4.6667, A 0.000, B 0.000, C 0.000 }
gfCNCPoint3[18800] = {X 357.0841, Y 26.7727, Z -4.6667, A 0.000, B 0.000, C 0.000 }
gfCNCPoint3[18801] = {X 357.1948, Y 25.0729, Z -4.6667, A 0.000, B 0.000, C 0.000 }
gfCNCPoint3[18802] = {X 357.1431, Y 23.3702, Z -4.6667, A 0.000, B 0.000, C 0.000 }
gfCNCPoint3[18803] = {X 356.9294, Y 21.6802, Z -4.6667, A 0.000, B 0.000, C 0.000 }
gfCNCPoint3[18804] = {X 356.5776, Y 20.1747, Z -4.6667, A 0.000, B 0.000, C 0.000 }
gfCNCPoint3[18805] = {X 356.0314, Y 18.7283, Z -4.6667, A 0.000, B 0.000, C 0.000 }
gfCNCPoint3[18806] = {X 355.3001, Y 17.3661, Z -4.6667, A 0.000, B 0.000, C 0.000 }
gfCNCPoint3[18807] = {X 354.3964, Y 16.1116, Z -4.6667, A 0.000, B 0.000, C 0.000 }
gfCNCPoint3[18808] = {X 353.5334, Y 15.1932, Z -4.6667, A 0.000, B 0.000, C 0.000 }
gfCNCPoint3[18809] = {X 352.5515, Y 14.4032, Z -4.6667, A 0.000, B 0.000, C 0.000 }
gfCNCPoint3[18810] = {X 351.4695, Y 13.7570, Z -4.6667, A 0.000, B 0.000, C 0.000 }
gfCNCPoint3[18811] = {X 350.3084, Y 13.2670, Z -4.6667, A 0.000, B 0.000, C 0.000 }
gfCNCPoint3[18812] = {X 349.0906, Y 12.9426, Z -4.6667, A 0.000, B 0.000, C 0.000 }
gfCNCPoint3[18813] = {X 347.3479, Y 12.7254, Z -4.6667, A 0.000, B 0.000, C 0.000 }
gfCNCPoint3[18814] = {X 345.5918, Y 12.7396, Z -4.6667, A 0.000, B 0.000, C 0.000 }
gfCNCPoint3[18815] = {X 343.8529, Y 12.9851, Z -4.6667, A 0.000, B 0.000, C 0.000 }
gfCNCPoint3[18816] = {X 342.1614, Y 13.4575, Z -4.6667, A 0.000, B 0.000, C 0.000 }
gfCNCPoint3[18817] = {X 340.5469, Y 14.1486, Z -4.6667, A 0.000, B 0.000, C 0.000 }
gfCNCPoint3[18818] = {X 339.0376, Y 15.0464, Z -4.6667, A 0.000, B 0.000, C 0.000 }
gfCNCPoint3[18819] = {X 338.9896, Y 15.9043, Z -4.6667, A 0.000, B 0.000, C 0.000 }
gfCNCPoint3[18820] = {X 338.7758, Y 16.7365, Z -4.6667, A 0.000, B 0.000, C 0.000 }
gfCNCPoint3[18821] = {X 338.4043, Y 17.5114, Z -4.6667, A 0.000, B 0.000, C 0.000 }
gfCNCPoint3[18822] = {X 337.8893, Y 18.1992, Z -4.6667, A 0.000, B 0.000, C 0.000 }
gfCNCPoint3[18823] = {X 337.2504, Y 18.7738, Z -4.6667, A 0.000, B 0.000, C 0.000 }
gfCNCPoint3[18824] = {X 336.5606, Y 19.2813, Z -4.6667, A 0.000, B 0.000, C 0.000 }
gfCNCPoint3[18825] = {X 335.7284, Y 19.7495, Z -4.6667, A 0.000, B 0.000, C 0.000 }
gfCNCPoint3[18826] = {X 334.8148, Y 20.0271, Z -4.6667, A 0.000, B 0.000, C 0.000 }
gfCNCPoint3[18827] = {X 333.8628, Y 20.1012, Z -4.6667, A 0.000, B 0.000, C 0.000 }
gfCNCPoint3[18828] = {X 332.9173, Y 19.9681, Z -4.6667, A 0.000, B 0.000, C 0.000 }
gfCNCPoint3[18829] = {X 332.0228, Y 19.6341, Z -4.6667, A 0.000, B 0.000, C 0.000 }
gfCNCPoint3[18830] = {X 331.2213, Y 19.1151, Z -4.6667, A 0.000, B 0.000, C 0.000 }
gfCNCPoint3[18831] = {X 330.5507, Y 18.4353, Z -4.6667, A 0.000, B 0.000, C 0.000 }
gfCNCPoint3[18832] = {X 330.0425, Y 17.6269, Z -4.6667, A 0.000, B 0.000, C 0.000 }
gfCNCPoint3[18833] = {X 326.5223, Y 10.3852, Z -4.6667, A 0.000, B 0.000, C 0.000 }
gfCNCPoint3[18834] = {X 326.2154, Y 9.5469, Z -4.6667, A 0.000, B 0.000, C 0.000 }
gfCNCPoint3[18835] = {X 326.0841, Y 8.6639, Z -4.6667, A 0.000, B 0.000, C 0.000 }
gfCNCPoint3[18836] = {X 326.1338, Y 7.7725, Z -4.6667, A 0.000, B 0.000, C 0.000 }
gfCNCPoint3[18837] = {X 326.3623, Y 6.9096, Z -4.6667, A 0.000, B 0.000, C 0.000 }
gfCNCPoint3[18838] = {X 326.7603, Y 6.1105, Z -4.6667, A 0.000, B 0.000, C 0.000 }
gfCNCPoint3[18839] = {X 327.3114, Y 5.4082, Z -4.6667, A 0.000, B 0.000, C 0.000 }
gfCNCPoint3[18840] = {X 327.9929, Y 4.8316, Z -4.6667, A 0.000, B 0.000, C 0.000 }
gfCNCPoint3[18841] = {X 328.6647, Y 4.3715, Z -4.6667, A 0.000, B 0.000, C 0.000 }
gfCNCPoint3[18842] = {X 329.5524, Y 3.9111, Z -4.6667, A 0.000, B 0.000, C 0.000 }
gfCNCPoint3[18843] = {X 330.5211, Y 3.6631, Z -4.6667, A 0.000, B 0.000, C 0.000 }
gfCNCPoint3[18844] = {X 331.5208, Y 3.6402, Z -4.6667, A 0.000, B 0.000, C 0.000 }
gfCNCPoint3[18845] = {X 332.4999, Y 3.8436, Z -4.6667, A 0.000, B 0.000, C 0.000 }
gfCNCPoint3[18846] = {X 333.5098, Y 3.2689, Z -4.6667, A 0.000, B 0.000, C 0.000 }
gfCNCPoint3[18847] = {X 334.5424, Y 2.7359, Z -4.6667, A 0.000, B 0.000, C 0.000 }
gfCNCPoint3[18848] = {X 334.3310, Y 2.3050, Z -4.6667, A 0.000, B 0.000, C 0.000 }
gfCNCPoint3[18849] = {X 2.3034, Y 2.3050, Z -4.6667, A 0.000, B 0.000, C 0.000 }
gfCNCPoint3[18850] = {X 2.3034, Y 6.8597, Z -4.6667, A 0.000, B 0.000, C 0.000 }
gfCNCPoint3[18851] = {X 2.3977, Y 6.8785, Z -4.6667, A 0.000, B 0.000, C 0.000 }
gfCNCPoint3[18852] = {X 2.8661, Y 6.6877, Z -4.6667, A 0.000, B 0.000, C 0.000 }
gfCNCPoint3[18853] = {X 3.3414, Y 6.5148, Z -4.6667, A 0.000, B 0.000, C 0.000 }
gfCNCPoint3[18854] = {X 5.4454, Y 5.7843, Z -4.6667, A 0.000, B 0.000, C 0.000 }
gfCNCPoint3[18855] = {X 7.6044, Y 5.2370, Z -4.6667, A 0.000, B 0.000, C 0.000 }
gfCNCPoint3[18856] = {X 9.8023, Y 4.8768, Z -4.6667, A 0.000, B 0.000, C 0.000 }
gfCNCPoint3[18857] = {X 12.0230, Y 4.7066, Z -4.6667, A 0.000, B 0.000, C 0.000 }
gfCNCPoint3[18858] = {X 14.2501, Y 4.7274, Z -4.6667, A 0.000, B 0.000, C 0.000 }
gfCNCPoint3[18859] = {X 16.4673, Y 4.9393, Z -4.6667, A 0.000, B 0.000, C 0.000 }
gfCNCPoint3[18860] = {X 18.0966, Y 5.2200, Z -4.6667, A 0.000, B 0.000, C 0.000 }
gfCNCPoint3[18861] = {X 19.6970, Y 5.6349, Z -4.6667, A 0.000, B 0.000, C 0.000 }
gfCNCPoint3[18862] = {X 21.2576, Y 6.1809, Z -4.6667, A 0.000, B 0.000, C 0.000 }
gfCNCPoint3[18863] = {X 22.7675, Y 6.8544, Z -4.6667, A 0.000, B 0.000, C 0.000 }
gfCNCPoint3[18864] = {X 24.4887, Y 7.8184, Z -4.6667, A 0.000, B 0.000, C 0.000 }
gfCNCPoint3[18865] = {X 26.1061, Y 8.9478, Z -4.6667, A 0.000, B 0.000, C 0.000 }
gfCNCPoint3[18866] = {X 27.4003, Y 10.0780, Z -4.6667, A 0.000, B 0.000, C 0.000 }
gfCNCPoint3[18867] = {X 28.5613, Y 11.3447, Z -4.6667, A 0.000, B 0.000, C 0.000 }
gfCNCPoint3[18868] = {X 29.5746, Y 12.7323, Z -4.6667, A 0.000, B 0.000, C 0.000 }
gfCNCPoint3[18869] = {X 30.4280, Y 14.2237, Z -4.6667, A 0.000, B 0.000, C 0.000 }
gfCNCPoint3[18870] = {X 31.1107, Y 15.8004, Z -4.6667, A 0.000, B 0.000, C 0.000 }
gfCNCPoint3[18871] = {X 31.6707, Y 17.7361, Z -4.6667, A 0.000, B 0.000, C 0.000 }
gfCNCPoint3[18872] = {X 32.0040, Y 19.7233, Z -4.6667, A 0.000, B 0.000, C 0.000 }
gfCNCPoint3[18873] = {X 32.1063, Y 21.7357, Z -4.6667, A 0.000, B 0.000, C 0.000 }
gfCNCPoint3[18874] = {X 31.9762, Y 23.7465, Z -4.6667, A 0.000, B 0.000, C 0.000 }
gfCNCPoint3[18875] = {X 31.6154, Y 25.7289, Z -4.6667, A 0.000, B 0.000, C 0.000 }
gfCNCPoint3[18876] = {X 31.1836, Y 27.1946, Z -4.6667, A 0.000, B 0.000, C 0.000 }
gfCNCPoint3[18877] = {X 30.5964, Y 28.6052, Z -4.6667, A 0.000, B 0.000, C 0.000 }
gfCNCPoint3[18878] = {X 29.8609, Y 29.9443, Z -4.6667, A 0.000, B 0.000, C 0.000 }
gfCNCPoint3[18879] = {X 29.4844, Y 30.5183, Z -4.6667, A 0.000, B 0.000, C 0.000 }
gfCNCPoint3[18880] = {X 29.0807, Y 31.0734, Z -4.6667, A 0.000, B 0.000, C 0.000 }
gfCNCPoint3[18881] = {X 29.6385, Y 31.7919, Z -4.6667, A 0.000, B 0.000, C 0.000 }
gfCNCPoint3[18882] = {X 30.0954, Y 32.5785, Z -4.6667, A 0.000, B 0.000, C 0.000 }
gfCNCPoint3[18883] = {X 33.1423, Y 38.8726, Z -4.6667, A 0.000, B 0.000, C 0.000 }
gfCNCPoint3[18884] = {X 33.5391, Y 39.8957, Z -4.6667, A 0.000, B 0.000, C 0.000 }
gfCNCPoint3[18885] = {X 33.7662, Y 40.9694, Z -4.6667, A 0.000, B 0.000, C 0.000 }
gfCNCPoint3[18886] = {X 33.8177, Y 42.0656, Z -4.6667, A 0.000, B 0.000, C 0.000 }
gfCNCPoint3[18887] = {X 33.7164, Y 43.0266, Z -4.6667, A 0.000, B 0.000, C 0.000 }
gfCNCPoint3[18888] = {X 33.4799, Y 43.9636, Z -4.6667, A 0.000, B 0.000, C 0.000 }
gfCNCPoint3[18889] = {X 33.1103, Y 44.8630, Z -4.6667, A 0.000, B 0.000, C 0.000 }
gfCNCPoint3[18890] = {X 32.6161, Y 45.7005, Z -4.6667, A 0.000, B 0.000, C 0.000 }
gfCNCPoint3[18891] = {X 32.0075, Y 46.4590, Z -4.6667, A 0.000, B 0.000, C 0.000 }
gfCNCPoint3[18892] = {X 31.2970, Y 47.1229, Z -4.6667, A 0.000, B 0.000, C 0.000 }
gfCNCPoint3[18893] = {X 30.7598, Y 47.5573, Z -4.6667, A 0.000, B 0.000, C 0.000 }
gfCNCPoint3[18894] = {X 29.8539, Y 48.1755, Z -4.6667, A 0.000, B 0.000, C 0.000 }
gfCNCPoint3[18895] = {X 28.8605, Y 48.6404, Z -4.6667, A 0.000, B 0.000, C 0.000 }
gfCNCPoint3[18896] = {X 27.8054, Y 48.9399, Z -4.6667, A 0.000, B 0.000, C 0.000 }
gfCNCPoint3[18897] = {X 26.7159, Y 49.0662, Z -4.6667, A 0.000, B 0.000, C 0.000 }
gfCNCPoint3[18898] = {X 25.6202, Y 49.0161, Z -4.6667, A 0.000, B 0.000, C 0.000 }
gfCNCPoint3[18899] = {X 23.9308, Y 49.8549, Z -4.6667, A 0.000, B 0.000, C 0.000 }
gfCNCPoint3[18900] = {X 22.1945, Y 50.5915, Z -4.6667, A 0.000, B 0.000, C 0.000 }
gfCNCPoint3[18901] = {X 20.4174, Y 51.2235, Z -4.6667, A 0.000, B 0.000, C 0.000 }
gfCNCPoint3[18902] = {X 18.2676, Y 51.8294, Z -4.6667, A 0.000, B 0.000, C 0.000 }
gfCNCPoint3[18903] = {X 16.0727, Y 52.2430, Z -4.6667, A 0.000, B 0.000, C 0.000 }
gfCNCPoint3[18904] = {X 13.8499, Y 52.4611, Z -4.6667, A 0.000, B 0.000, C 0.000 }
gfCNCPoint3[18905] = {X 11.6164, Y 52.4820, Z -4.6667, A 0.000, B 0.000, C 0.000 }
gfCNCPoint3[18906] = {X 9.3899, Y 52.3056, Z -4.6667, A 0.000, B 0.000, C 0.000 }
gfCNCPoint3[18907] = {X 7.1877, Y 51.9331, Z -4.6667, A 0.000, B 0.000, C 0.000 }
gfCNCPoint3[18908] = {X 6.2989, Y 51.7229, Z -4.6667, A 0.000, B 0.000, C 0.000 }
gfCNCPoint3[18909] = {X 5.4212, Y 51.4706, Z -4.6667, A 0.000, B 0.000, C 0.000 }
gfCNCPoint3[18910] = {X 3.8339, Y 50.8952, Z -4.6667, A 0.000, B 0.000, C 0.000 }
gfCNCPoint3[18911] = {X 2.3034, Y 50.1825, Z -4.6667, A 0.000, B 0.000, C 0.000 }
gfCNCPoint3[18912] = {X 2.3034, Y 97.6950, Z -4.6667, A 0.000, B 0.000, C 0.000 }
gfCNCPoint3[18913] = {X 120.1200, Y 97.6950, Z -4.6667, A 0.000, B 0.000, C 0.000 }
gfCNCPoint3[18914] = {X 120.1200, Y 97.0659, Z -4.6667, A 0.000, B 0.000, C 0.000 }
gfCNCPoint3[18915] = {X 120.2338, Y 96.0181, Z -4.6667, A 0.000, B 0.000, C 0.000 }
gfCNCPoint3[18916] = {X 120.5700, Y 95.0191, Z -4.6667, A 0.000, B 0.000, C 0.000 }
gfCNCPoint3[18917] = {X 121.1128, Y 94.1156, Z -4.6667, A 0.000, B 0.000, C 0.000 }
gfCNCPoint3[18918] = {X 121.8370, Y 93.3498, Z -4.6667, A 0.000, B 0.000, C 0.000 }
gfCNCPoint3[18919] = {X 122.7087, Y 92.7573, Z -4.6667, A 0.000, B 0.000, C 0.000 }
gfCNCPoint3[18920] = {X 123.6873, Y 92.3658, Z -4.6667, A 0.000, B 0.000, C 0.000 }
gfCNCPoint3[18921] = {X 124.7272, Y 92.1936, Z -4.6667, A 0.000, B 0.000, C 0.000 }
gfCNCPoint3[18922] = {X 124.7860, Y 92.1785, Z -4.6667, A 0.000, B 0.000, C 0.000 }
gfCNCPoint3[18923] = {X 124.8457, Y 92.1675, Z -4.6667, A 0.000, B 0.000, C 0.000 }
gfCNCPoint3[18924] = {X 125.3649, Y 92.0905, Z -4.6667, A 0.000, B 0.000, C 0.000 }
gfCNCPoint3[18925] = {X 126.0998, Y 91.9694, Z -4.6667, A 0.000, B 0.000, C 0.000 }
gfCNCPoint3[18926] = {X 126.8255, Y 91.8020, Z -4.6667, A 0.000, B 0.000, C 0.000 }
gfCNCPoint3[18927] = {X 127.9734, Y 90.7129, Z -4.6667, A 0.000, B 0.000, C 0.000 }
gfCNCPoint3[18928] = {X 129.0629, Y 89.5654, Z -4.6667, A 0.000, B 0.000, C 0.000 }
gfCNCPoint3[18929] = {X 154.9460, Y 61.1420, Z -4.6667, A 0.000, B 0.000, C 0.000 }
gfCNCPoint3[18930] = {X 154.6592, Y 60.4495, Z -4.6667, A 0.000, B 0.000, C 0.000 }
gfCNCPoint3[18931] = {X 154.4819, Y 59.7212, Z -4.6667, A 0.000, B 0.000, C 0.000 }
gfCNCPoint3[18932] = {X 154.4181, Y 58.9744, Z -4.6667, A 0.000, B 0.000, C 0.000 }
gfCNCPoint3[18933] = {X 154.4180, Y 58.0000, Z -4.6667, A 0.000, B 0.000, C 0.000 }
gfCNCPoint3[18934] = {X 154.5117, Y 57.0480, Z -4.6667, A 0.000, B 0.000, C 0.000 }
gfCNCPoint3[18935] = {X 154.7894, Y 56.1325, Z -4.6667, A 0.000, B 0.000, C 0.000 }
gfCNCPoint3[18936] = {X 155.2404, Y 55.2888, Z -4.6667, A 0.000, B 0.000, C 0.000 }
gfCNCPoint3[18937] = {X 155.8473, Y 54.5493, Z -4.6667, A 0.000, B 0.000, C 0.000 }
gfCNCPoint3[18938] = {X 156.5868, Y 53.9424, Z -4.6667, A 0.000, B 0.000, C 0.000 }
gfCNCPoint3[18939] = {X 157.4305, Y 53.4915, Z -4.6667, A 0.000, B 0.000, C 0.000 }
gfCNCPoint3[18940] = {X 158.3459, Y 53.2138, Z -4.6667, A 0.000, B 0.000, C 0.000 }
gfCNCPoint3[18941] = {X 159.2980, Y 53.1200, Z -4.6667, A 0.000, B 0.000, C 0.000 }
gfCNCPoint3[18942] = {X 178.5335, Y 53.1200, Z -4.6667, A 0.000, B 0.000, C 0.000 }
gfCNCPoint3[18943] = {X 179.4855, Y 53.2138, Z -4.6667, A 0.000, B 0.000, C 0.000 }
gfCNCPoint3[18944] = {X 180.4010, Y 53.4915, Z -4.6667, A 0.000, B 0.000, C 0.000 }
gfCNCPoint3[18945] = {X 181.2447, Y 53.9424, Z -4.6667, A 0.000, B 0.000, C 0.000 }
gfCNCPoint3[18946] = {X 181.9842, Y 54.5493, Z -4.6667, A 0.000, B 0.000, C 0.000 }
gfCNCPoint3[18947] = {X 182.5911, Y 55.2888, Z -4.6667, A 0.000, B 0.000, C 0.000 }
gfCNCPoint3[18948] = {X 183.0420, Y 56.1325, Z -4.6667, A 0.000, B 0.000, C 0.000 }
gfCNCPoint3[18949] = {X 183.3197, Y 57.0480, Z -4.6667, A 0.000, B 0.000, C 0.000 }
gfCNCPoint3[18950] = {X 183.4135, Y 58.0000, Z -4.6667, A 0.000, B 0.000, C 0.000 }
gfCNCPoint3[18951] = {X 183.4133, Y 58.9744, Z -4.6667, A 0.000, B 0.000, C 0.000 }
gfCNCPoint3[18952] = {X 183.3512, Y 59.7112, Z -4.6667, A 0.000, B 0.000, C 0.000 }
gfCNCPoint3[18953] = {X 183.1785, Y 60.4303, Z -4.6667, A 0.000, B 0.000, C 0.000 }
gfCNCPoint3[18954] = {X 182.8991, Y 61.1149, Z -4.6667, A 0.000, B 0.000, C 0.000 }
gfCNCPoint3[18955] = {X 209.8917, Y 90.5758, Z -4.6667, A 0.000, B 0.000, C 0.000 }
gfCNCPoint3[18956] = {X 210.5202, Y 91.2135, Z -4.6667, A 0.000, B 0.000, C 0.000 }
gfCNCPoint3[18957] = {X 211.1934, Y 91.8037, Z -4.6667, A 0.000, B 0.000, C 0.000 }
gfCNCPoint3[18958] = {X 211.3595, Y 91.9082, Z -4.6667, A 0.000, B 0.000, C 0.000 }
gfCNCPoint3[18959] = {X 211.5461, Y 91.9693, Z -4.6667, A 0.000, B 0.000, C 0.000 }
gfCNCPoint3[18960] = {X 212.2018, Y 92.1095, Z -4.6667, A 0.000, B 0.000, C 0.000 }
gfCNCPoint3[18961] = {X 213.4083, Y 92.2615, Z -4.6667, A 0.000, B 0.000, C 0.000 }
gfCNCPoint3[18962] = {X 214.4425, Y 92.1753, Z -4.6667, A 0.000, B 0.000, C 0.000 }
gfCNCPoint3[18963] = {X 215.4785, Y 92.1163, Z -4.6667, A 0.000, B 0.000, C 0.000 }
gfCNCPoint3[18964] = {X 216.0525, Y 92.0566, Z -4.6667, A 0.000, B 0.000, C 0.000 }
gfCNCPoint3[18965] = {X 216.6054, Y 91.8913, Z -4.6667, A 0.000, B 0.000, C 0.000 }
gfCNCPoint3[18966] = {X 217.1180, Y 91.6261, Z -4.6667, A 0.000, B 0.000, C 0.000 }
gfCNCPoint3[18967] = {X 244.6009, Y 74.0196, Z -4.6667, A 0.000, B 0.000, C 0.000 }
gfCNCPoint3[18968] = {X 221.4278, Y 64.9258, Z -4.6667, A 0.000, B 0.000, C 0.000 }
gfCNCPoint3[18969] = {X 219.7199, Y 64.3535, Z -4.6667, A 0.000, B 0.000, C 0.000 }
gfCNCPoint3[18970] = {X 217.9578, Y 63.9803, Z -4.6667, A 0.000, B 0.000, C 0.000 }
gfCNCPoint3[18971] = {X 216.1645, Y 63.8112, Z -4.6667, A 0.000, B 0.000, C 0.000 }
gfCNCPoint3[18972] = {X 215.1119, Y 63.6594, Z -4.6667, A 0.000, B 0.000, C 0.000 }
gfCNCPoint3[18973] = {X 214.1173, Y 63.2832, Z -4.6667, A 0.000, B 0.000, C 0.000 }
gfCNCPoint3[18974] = {X 213.2277, Y 62.7004, Z -4.6667, A 0.000, B 0.000, C 0.000 }
gfCNCPoint3[18975] = {X 212.4856, Y 61.9388, Z -4.6667, A 0.000, B 0.000, C 0.000 }
gfCNCPoint3[18976] = {X 211.9260, Y 61.0345, Z -4.6667, A 0.000, B 0.000, C 0.000 }
gfCNCPoint3[18977] = {X 211.5756, Y 60.0305, Z -4.6667, A 0.000, B 0.000, C 0.000 }
gfCNCPoint3[18978] = {X 211.4510, Y 58.9744, Z -4.6667, A 0.000, B 0.000, C 0.000 }
gfCNCPoint3[18979] = {X 211.4508, Y 58.0000, Z -4.6667, A 0.000, B 0.000, C 0.000 }
gfCNCPoint3[18980] = {X 211.5446, Y 57.0480, Z -4.6667, A 0.000, B 0.000, C 0.000 }
gfCNCPoint3[18981] = {X 211.8223, Y 56.1325, Z -4.6667, A 0.000, B 0.000, C 0.000 }
gfCNCPoint3[18982] = {X 212.2732, Y 55.2888, Z -4.6667, A 0.000, B 0.000, C 0.000 }
gfCNCPoint3[18983] = {X 212.8801, Y 54.5493, Z -4.6667, A 0.000, B 0.000, C 0.000 }
gfCNCPoint3[18984] = {X 213.6196, Y 53.9424, Z -4.6667, A 0.000, B 0.000, C 0.000 }
gfCNCPoint3[18985] = {X 214.4633, Y 53.4915, Z -4.6667, A 0.000, B 0.000, C 0.000 }
gfCNCPoint3[18986] = {X 215.3788, Y 53.2138, Z -4.6667, A 0.000, B 0.000, C 0.000 }
gfCNCPoint3[18987] = {X 216.3308, Y 53.1200, Z -4.6667, A 0.000, B 0.000, C 0.000 }
gfCNCPoint3[18988] = {X 237.2617, Y 53.1200, Z -4.6667, A 0.000, B 0.000, C 0.000 }
gfCNCPoint3[18989] = {X 238.3265, Y 53.2376, Z -4.6667, A 0.000, B 0.000, C 0.000 }
gfCNCPoint3[18990] = {X 239.3400, Y 53.5847, Z -4.6667, A 0.000, B 0.000, C 0.000 }
gfCNCPoint3[18991] = {X 240.2533, Y 54.1446, Z -4.6667, A 0.000, B 0.000, C 0.000 }
gfCNCPoint3[18992] = {X 241.0225, Y 54.8902, Z -4.6667, A 0.000, B 0.000, C 0.000 }
gfCNCPoint3[18993] = {X 241.6104, Y 55.7858, Z -4.6667, A 0.000, B 0.000, C 0.000 }
gfCNCPoint3[18994] = {X 241.9888, Y 56.7880, Z -4.6667, A 0.000, B 0.000, C 0.000 }
gfCNCPoint3[18995] = {X 242.1393, Y 57.8487, Z -4.6667, A 0.000, B 0.000, C 0.000 }
gfCNCPoint3[18996] = {X 248.3213, Y 60.2592, Z -4.6667, A 0.000, B 0.000, C 0.000 }
gfCNCPoint3[18997] = {X 275.0727, Y 70.8773, Z -4.6667, A 0.000, B 0.000, C 0.000 }
gfCNCPoint3[18998] = {X 275.0723, Y 63.6741, Z -4.6667, A 0.000, B 0.000, C 0.000 }
gfCNCPoint3[18999] = {X 274.0641, Y 63.3057, Z -4.6667, A 0.000, B 0.000, C 0.000 }
gfCNCPoint3[19000] = {X 273.1608, Y 62.7259, Z -4.6667, A 0.000, B 0.000, C 0.000 }
gfCNCPoint3[19001] = {X 272.4061, Y 61.9625, Z -4.6667, A 0.000, B 0.000, C 0.000 }
gfCNCPoint3[19002] = {X 271.8366, Y 61.0526, Z -4.6667, A 0.000, B 0.000, C 0.000 }
gfCNCPoint3[19003] = {X 271.4797, Y 60.0403, Z -4.6667, A 0.000, B 0.000, C 0.000 }
gfCNCPoint3[19004] = {X 271.3529, Y 58.9744, Z -4.6667, A 0.000, B 0.000, C 0.000 }
gfCNCPoint3[19005] = {X 271.3527, Y 58.0000, Z -4.6667, A 0.000, B 0.000, C 0.000 }
gfCNCPoint3[19006] = {X 271.4465, Y 57.0480, Z -4.6667, A 0.000, B 0.000, C 0.000 }
gfCNCPoint3[19007] = {X 271.7242, Y 56.1325, Z -4.6667, A 0.000, B 0.000, C 0.000 }
gfCNCPoint3[19008] = {X 272.1751, Y 55.2888, Z -4.6667, A 0.000, B 0.000, C 0.000 }
gfCNCPoint3[19009] = {X 272.7820, Y 54.5493, Z -4.6667, A 0.000, B 0.000, C 0.000 }
gfCNCPoint3[19010] = {X 273.5215, Y 53.9424, Z -4.6667, A 0.000, B 0.000, C 0.000 }
gfCNCPoint3[19011] = {X 274.3652, Y 53.4915, Z -4.6667, A 0.000, B 0.000, C 0.000 }
gfCNCPoint3[19012] = {X 275.2806, Y 53.2138, Z -4.6667, A 0.000, B 0.000, C 0.000 }
gfCNCPoint3[19013] = {X 276.2327, Y 53.1200, Z -4.6667, A 0.000, B 0.000, C 0.000 }
gfCNCPoint3[19014] = {X 292.7731, Y 53.1200, Z -4.6667, A 0.000, B 0.000, C 0.000 }
gfCNCPoint3[19015] = {X 293.7251, Y 53.2138, Z -4.6667, A 0.000, B 0.000, C 0.000 }
gfCNCPoint3[19016] = {X 294.6406, Y 53.4915, Z -4.6667, A 0.000, B 0.000, C 0.000 }
gfCNCPoint3[19017] = {X 295.4843, Y 53.9424, Z -4.6667, A 0.000, B 0.000, C 0.000 }
gfCNCPoint3[19018] = {X 296.2238, Y 54.5493, Z -4.6667, A 0.000, B 0.000, C 0.000 }
gfCNCPoint3[19019] = {X 296.8307, Y 55.2888, Z -4.6667, A 0.000, B 0.000, C 0.000 }
gfCNCPoint3[19020] = {X 297.2816, Y 56.1325, Z -4.6667, A 0.000, B 0.000, C 0.000 }
gfCNCPoint3[19021] = {X 297.5593, Y 57.0480, Z -4.6667, A 0.000, B 0.000, C 0.000 }
gfCNCPoint3[19022] = {X 297.6531, Y 58.0000, Z -4.6667, A 0.000, B 0.000, C 0.000 }
gfCNCPoint3[19023] = {X 297.6531, Y 58.9369, Z -4.6667, A 0.000, B 0.000, C 0.000 }
gfCNCPoint3[19024] = {X 297.5308, Y 60.0091, Z -4.6667, A 0.000, B 0.000, C 0.000 }
gfCNCPoint3[19025] = {X 297.1766, Y 61.0285, Z -4.6667, A 0.000, B 0.000, C 0.000 }
gfCNCPoint3[19026] = {X 296.6077, Y 61.9456, Z -4.6667, A 0.000, B 0.000, C 0.000 }
gfCNCPoint3[19027] = {X 295.8517, Y 62.7158, Z -4.6667, A 0.000, B 0.000, C 0.000 }
gfCNCPoint3[19028] = {X 294.9454, Y 63.3016, Z -4.6667, A 0.000, B 0.000, C 0.000 }
gfCNCPoint3[19029] = {X 293.9328, Y 63.6747, Z -4.6667, A 0.000, B 0.000, C 0.000 }
gfCNCPoint3[19030] = {X 293.9328, Y 92.3201, Z -4.6667, A 0.000, B 0.000, C 0.000 }
gfCNCPoint3[19031] = {X 294.9452, Y 92.6958, Z -4.6667, A 0.000, B 0.000, C 0.000 }
gfCNCPoint3[19032] = {X 295.8512, Y 93.2836, Z -4.6667, A 0.000, B 0.000, C 0.000 }
gfCNCPoint3[19033] = {X 296.6068, Y 94.0551, Z -4.6667, A 0.000, B 0.000, C 0.000 }
gfCNCPoint3[19034] = {X 297.1756, Y 94.9731, Z -4.6667, A 0.000, B 0.000, C 0.000 }
gfCNCPoint3[19035] = {X 297.5301, Y 95.9932, Z -4.6667, A 0.000, B 0.000, C 0.000 }
gfCNCPoint3[19036] = {X 297.6531, Y 97.0661, Z -4.6667, A 0.000, B 0.000, C 0.000 }
gfCNCPoint3[19037] = {X 297.6531, Y 97.6950, Z -4.6667, A 0.000, B 0.000, C 0.000 }
gfCNCPoint3[19038] = {X 297.1731, Y 97.6950, Z -4.6667, A 0.000, B 0.000, C 0.000 }
gfCNCPoint3[19039] = {X 297.1731, Y 98.0000, Z -4.6667, A 0.000, B 0.000, C 0.000 }
gfCNCPoint3[19040] = {X 297.0628, Y 98.9791, Z -4.6667, A 0.000, B 0.000, C 0.000 }
gfCNCPoint3[19041] = {X 296.7373, Y 99.9091, Z -4.6667, A 0.000, B 0.000, C 0.000 }
gfCNCPoint3[19042] = {X 296.2131, Y 100.7434, Z -4.6667, A 0.000, B 0.000, C 0.000 }
gfCNCPoint3[19043] = {X 295.5164, Y 101.4401, Z -4.6667, A 0.000, B 0.000, C 0.000 }
gfCNCPoint3[19044] = {X 294.6822, Y 101.9643, Z -4.6667, A 0.000, B 0.000, C 0.000 }
gfCNCPoint3[19045] = {X 293.7522, Y 102.2897, Z -4.6667, A 0.000, B 0.000, C 0.000 }
gfCNCPoint3[19046] = {X 292.7731, Y 102.4000, Z -4.6667, A 0.000, B 0.000, C 0.000 }
gfCNCPoint3[19047] = {X 276.2327, Y 102.4000, Z -4.6667, A 0.000, B 0.000, C 0.000 }
gfCNCPoint3[19048] = {X 275.2536, Y 102.2897, Z -4.6667, A 0.000, B 0.000, C 0.000 }
gfCNCPoint3[19049] = {X 274.3236, Y 101.9643, Z -4.6667, A 0.000, B 0.000, C 0.000 }
gfCNCPoint3[19050] = {X 273.4893, Y 101.4401, Z -4.6667, A 0.000, B 0.000, C 0.000 }
gfCNCPoint3[19051] = {X 272.7926, Y 100.7434, Z -4.6667, A 0.000, B 0.000, C 0.000 }
gfCNCPoint3[19052] = {X 272.2684, Y 99.9091, Z -4.6667, A 0.000, B 0.000, C 0.000 }
gfCNCPoint3[19053] = {X 271.9430, Y 98.9791, Z -4.6667, A 0.000, B 0.000, C 0.000 }
gfCNCPoint3[19054] = {X 271.8327, Y 98.0000, Z -4.6667, A 0.000, B 0.000, C 0.000 }
gfCNCPoint3[19055] = {X 271.8329, Y 97.0190, Z -4.6667, A 0.000, B 0.000, C 0.000 }
gfCNCPoint3[19056] = {X 271.9305, Y 96.1432, Z -4.6667, A 0.000, B 0.000, C 0.000 }
gfCNCPoint3[19057] = {X 272.2006, Y 95.3045, Z -4.6667, A 0.000, B 0.000, C 0.000 }
gfCNCPoint3[19058] = {X 272.6325, Y 94.5364, Z -4.6667, A 0.000, B 0.000, C 0.000 }
gfCNCPoint3[19059] = {X 273.2087, Y 93.8698, Z -4.6667, A 0.000, B 0.000, C 0.000 }
gfCNCPoint3[19060] = {X 273.9062, Y 93.3313, Z -4.6667, A 0.000, B 0.000, C 0.000 }
gfCNCPoint3[19061] = {X 274.6970, Y 92.9426, Z -4.6667, A 0.000, B 0.000, C 0.000 }
gfCNCPoint3[19062] = {X 275.5494, Y 92.7193, Z -4.6667, A 0.000, B 0.000, C 0.000 }
gfCNCPoint3[19063] = {X 275.5494, Y 85.6495, Z -4.6667, A 0.000, B 0.000, C 0.000 }
gfCNCPoint3[19064] = {X 262.6481, Y 80.5922, Z -4.6667, A 0.000, B 0.000, C 0.000 }
gfCNCPoint3[19065] = {X 262.3201, Y 80.7990, Z -4.6667, A 0.000, B 0.000, C 0.000 }
gfCNCPoint3[19066] = {X 237.8769, Y 96.6315, Z -4.6667, A 0.000, B 0.000, C 0.000 }
gfCNCPoint3[19067] = {X 237.8798, Y 97.0659, Z -4.6667, A 0.000, B 0.000, C 0.000 }
gfCNCPoint3[19068] = {X 237.8798, Y 98.0000, Z -4.6667, A 0.000, B 0.000, C 0.000 }
gfCNCPoint3[19069] = {X 237.7695, Y 98.9791, Z -4.6667, A 0.000, B 0.000, C 0.000 }
gfCNCPoint3[19070] = {X 237.4440, Y 99.9091, Z -4.6667, A 0.000, B 0.000, C 0.000 }
gfCNCPoint3[19071] = {X 236.9198, Y 100.7434, Z -4.6667, A 0.000, B 0.000, C 0.000 }
gfCNCPoint3[19072] = {X 236.2231, Y 101.4401, Z -4.6667, A 0.000, B 0.000, C 0.000 }
gfCNCPoint3[19073] = {X 235.3889, Y 101.9643, Z -4.6667, A 0.000, B 0.000, C 0.000 }
gfCNCPoint3[19074] = {X 234.4589, Y 102.2897, Z -4.6667, A 0.000, B 0.000, C 0.000 }
gfCNCPoint3[19075] = {X 233.4798, Y 102.4000, Z -4.6667, A 0.000, B 0.000, C 0.000 }
gfCNCPoint3[19076] = {X 214.1790, Y 102.4000, Z -4.6667, A 0.000, B 0.000, C 0.000 }
gfCNCPoint3[19077] = {X 213.7862, Y 102.3824, Z -4.6667, A 0.000, B 0.000, C 0.000 }
gfCNCPoint3[19078] = {X 213.3966, Y 102.3299, Z -4.6667, A 0.000, B 0.000, C 0.000 }
gfCNCPoint3[19079] = {X 213.0069, Y 102.3824, Z -4.6667, A 0.000, B 0.000, C 0.000 }
gfCNCPoint3[19080] = {X 212.6141, Y 102.4000, Z -4.6667, A 0.000, B 0.000, C 0.000 }
gfCNCPoint3[19081] = {X 194.9870, Y 102.4000, Z -4.6667, A 0.000, B 0.000, C 0.000 }
gfCNCPoint3[19082] = {X 194.0079, Y 102.2897, Z -4.6667, A 0.000, B 0.000, C 0.000 }
gfCNCPoint3[19083] = {X 193.0779, Y 101.9643, Z -4.6667, A 0.000, B 0.000, C 0.000 }
gfCNCPoint3[19084] = {X 192.2436, Y 101.4401, Z -4.6667, A 0.000, B 0.000, C 0.000 }
gfCNCPoint3[19085] = {X 191.5469, Y 100.7434, Z -4.6667, A 0.000, B 0.000, C 0.000 }
gfCNCPoint3[19086] = {X 191.0227, Y 99.9091, Z -4.6667, A 0.000, B 0.000, C 0.000 }
gfCNCPoint3[19087] = {X 190.6973, Y 98.9791, Z -4.6667, A 0.000, B 0.000, C 0.000 }
gfCNCPoint3[19088] = {X 190.5870, Y 98.0000, Z -4.6667, A 0.000, B 0.000, C 0.000 }
gfCNCPoint3[19089] = {X 190.5870, Y 97.0659, Z -4.6667, A 0.000, B 0.000, C 0.000 }
gfCNCPoint3[19090] = {X 190.6897, Y 96.1207, Z -4.6667, A 0.000, B 0.000, C 0.000 }
gfCNCPoint3[19091] = {X 190.9931, Y 95.2196, Z -4.6667, A 0.000, B 0.000, C 0.000 }
gfCNCPoint3[19092] = {X 191.4830, Y 94.4047, Z -4.6667, A 0.000, B 0.000, C 0.000 }
gfCNCPoint3[19093] = {X 188.5295, Y 91.1802, Z -4.6667, A 0.000, B 0.000, C 0.000 }
gfCNCPoint3[19094] = {X 150.1254, Y 91.1802, Z -4.6667, A 0.000, B 0.000, C 0.000 }
gfCNCPoint3[19095] = {X 147.2496, Y 94.3662, Z -4.6667, A 0.000, B 0.000, C 0.000 }
gfCNCPoint3[19096] = {X 147.7556, Y 95.1905, Z -4.6667, A 0.000, B 0.000, C 0.000 }
gfCNCPoint3[19097] = {X 148.0704, Y 96.1050, Z -4.6667, A 0.000, B 0.000, C 0.000 }
gfCNCPoint3[19098] = {X 148.1791, Y 97.0661, Z -4.6667, A 0.000, B 0.000, C 0.000 }
gfCNCPoint3[19099] = {X 148.1791, Y 98.0000, Z -4.6667, A 0.000, B 0.000, C 0.000 }
gfCNCPoint3[19100] = {X 148.0688, Y 98.9791, Z -4.6667, A 0.000, B 0.000, C 0.000 }
gfCNCPoint3[19101] = {X 147.7434, Y 99.9091, Z -4.6667, A 0.000, B 0.000, C 0.000 }
gfCNCPoint3[19102] = {X 147.2192, Y 100.7434, Z -4.6667, A 0.000, B 0.000, C 0.000 }
gfCNCPoint3[19103] = {X 146.5225, Y 101.4401, Z -4.6667, A 0.000, B 0.000, C 0.000 }
gfCNCPoint3[19104] = {X 145.6882, Y 101.9643, Z -4.6667, A 0.000, B 0.000, C 0.000 }
gfCNCPoint3[19105] = {X 144.7582, Y 102.2897, Z -4.6667, A 0.000, B 0.000, C 0.000 }
gfCNCPoint3[19106] = {X 143.7791, Y 102.4000, Z -4.6667, A 0.000, B 0.000, C 0.000 }
gfCNCPoint3[19107] = {X 125.0000, Y 102.4000, Z -4.6667, A 0.000, B 0.000, C 0.000 }
gfCNCPoint3[19108] = {X 124.0209, Y 102.2897, Z -4.6667, A 0.000, B 0.000, C 0.000 }
gfCNCPoint3[19109] = {X 123.0909, Y 101.9643, Z -4.6667, A 0.000, B 0.000, C 0.000 }
gfCNCPoint3[19110] = {X 122.2566, Y 101.4401, Z -4.6667, A 0.000, B 0.000, C 0.000 }
gfCNCPoint3[19111] = {X 121.5599, Y 100.7434, Z -4.6667, A 0.000, B 0.000, C 0.000 }
gfCNCPoint3[19112] = {X 121.0357, Y 99.9091, Z -4.6667, A 0.000, B 0.000, C 0.000 }
gfCNCPoint3[19113] = {X 120.7103, Y 98.9791, Z -4.6667, A 0.000, B 0.000, C 0.000 }
gfCNCPoint3[19114] = {X 120.6000, Y 98.0000, Z -4.6667, A 0.000, B 0.000, C 0.000 }
gfCNCPoint3[19115] = {X 120.6000, Y 97.0659, Z -4.6667, A 0.000, B 0.000, C 0.000 }
gfCNCPoint3[19116] = {X 120.7046, Y 96.1121, Z -4.6667, A 0.000, B 0.000, C 0.000 }
gfCNCPoint3[19117] = {X 121.0135, Y 95.2036, Z -4.6667, A 0.000, B 0.000, C 0.000 }
gfCNCPoint3[19118] = {X 121.5121, Y 94.3837, Z -4.6667, A 0.000, B 0.000, C 0.000 }
gfCNCPoint3[19119] = {X 122.1765, Y 93.6914, Z -4.6667, A 0.000, B 0.000, C 0.000 }
gfCNCPoint3[19120] = {X 122.9751, Y 93.1595, Z -4.6667, A 0.000, B 0.000, C 0.000 }
gfCNCPoint3[19121] = {X 123.8701, Y 92.8135, Z -4.6667, A 0.000, B 0.000, C 0.000 }
gfCNCPoint3[19122] = {X 124.8188, Y 92.6697, Z -4.6667, A 0.000, B 0.000, C 0.000 }
gfCNCPoint3[19123] = {X 124.8666, Y 92.6529, Z -4.6667, A 0.000, B 0.000, C 0.000 }
gfCNCPoint3[19124] = {X 124.9161, Y 92.6423, Z -4.6667, A 0.000, B 0.000, C 0.000 }
gfCNCPoint3[19125] = {X 125.4412, Y 92.5645, Z -4.6667, A 0.000, B 0.000, C 0.000 }
gfCNCPoint3[19126] = {X 126.2566, Y 92.4275, Z -4.6667, A 0.000, B 0.000, C 0.000 }
gfCNCPoint3[19127] = {X 127.0608, Y 92.2357, Z -4.6667, A 0.000, B 0.000, C 0.000 }
gfCNCPoint3[19128] = {X 128.2726, Y 91.0924, Z -4.6667, A 0.000, B 0.000, C 0.000 }
gfCNCPoint3[19129] = {X 129.4207, Y 89.8854, Z -4.6667, A 0.000, B 0.000, C 0.000 }
gfCNCPoint3[19130] = {X 133.5081, Y 85.3891, Z -4.6667, A 0.000, B 0.000, C 0.000 }
gfCNCPoint3[19131] = {X 155.5327, Y 61.2107, Z -4.6667, A 0.000, B 0.000, C 0.000 }
gfCNCPoint3[19132] = {X 155.1840, Y 60.4946, Z -4.6667, A 0.000, B 0.000, C 0.000 }
gfCNCPoint3[19133] = {X 154.9701, Y 59.7273, Z -4.6667, A 0.000, B 0.000, C 0.000 }
gfCNCPoint3[19134] = {X 154.8980, Y 58.9340, Z -4.6667, A 0.000, B 0.000, C 0.000 }
gfCNCPoint3[19135] = {X 154.8980, Y 58.0000, Z -4.6667, A 0.000, B 0.000, C 0.000 }
gfCNCPoint3[19136] = {X 155.0083, Y 57.0209, Z -4.6667, A 0.000, B 0.000, C 0.000 }
gfCNCPoint3[19137] = {X 155.3337, Y 56.0909, Z -4.6667, A 0.000, B 0.000, C 0.000 }
gfCNCPoint3[19138] = {X 155.8579, Y 55.2566, Z -4.6667, A 0.000, B 0.000, C 0.000 }
gfCNCPoint3[19139] = {X 156.5546, Y 54.5599, Z -4.6667, A 0.000, B 0.000, C 0.000 }
gfCNCPoint3[19140] = {X 157.3889, Y 54.0357, Z -4.6667, A 0.000, B 0.000, C 0.000 }
gfCNCPoint3[19141] = {X 158.3189, Y 53.7103, Z -4.6667, A 0.000, B 0.000, C 0.000 }
gfCNCPoint3[19142] = {X 159.2980, Y 53.6000, Z -4.6667, A 0.000, B 0.000, C 0.000 }
gfCNCPoint3[19143] = {X 178.5335, Y 53.6000, Z -4.6667, A 0.000, B 0.000, C 0.000 }
gfCNCPoint3[19144] = {X 179.5126, Y 53.7103, Z -4.6667, A 0.000, B 0.000, C 0.000 }
gfCNCPoint3[19145] = {X 180.4426, Y 54.0357, Z -4.6667, A 0.000, B 0.000, C 0.000 }
gfCNCPoint3[19146] = {X 181.2769, Y 54.5599, Z -4.6667, A 0.000, B 0.000, C 0.000 }
gfCNCPoint3[19147] = {X 181.9736, Y 55.2566, Z -4.6667, A 0.000, B 0.000, C 0.000 }
gfCNCPoint3[19148] = {X 182.4978, Y 56.0909, Z -4.6667, A 0.000, B 0.000, C 0.000 }
gfCNCPoint3[19149] = {X 182.8232, Y 57.0209, Z -4.6667, A 0.000, B 0.000, C 0.000 }
gfCNCPoint3[19150] = {X 182.9335, Y 58.0000, Z -4.6667, A 0.000, B 0.000, C 0.000 }
gfCNCPoint3[19151] = {X 182.9334, Y 58.9704, Z -4.6667, A 0.000, B 0.000, C 0.000 }
gfCNCPoint3[19152] = {X 182.8587, Y 59.7418, Z -4.6667, A 0.000, B 0.000, C 0.000 }
gfCNCPoint3[19153] = {X 182.6499, Y 60.4881, Z -4.6667, A 0.000, B 0.000, C 0.000 }
gfCNCPoint3[19154] = {X 182.3134, Y 61.1862, Z -4.6667, A 0.000, B 0.000, C 0.000 }
gfCNCPoint3[19155] = {X 209.5378, Y 90.9001, Z -4.6667, A 0.000, B 0.000, C 0.000 }
gfCNCPoint3[19156] = {X 210.1908, Y 91.5627, Z -4.6667, A 0.000, B 0.000, C 0.000 }
gfCNCPoint3[19157] = {X 210.8903, Y 92.1759, Z -4.6667, A 0.000, B 0.000, C 0.000 }
gfCNCPoint3[19158] = {X 211.1521, Y 92.3410, Z -4.6667, A 0.000, B 0.000, C 0.000 }
gfCNCPoint3[19159] = {X 211.4457, Y 92.4387, Z -4.6667, A 0.000, B 0.000, C 0.000 }
gfCNCPoint3[19160] = {X 212.1215, Y 92.5831, Z -4.6667, A 0.000, B 0.000, C 0.000 }
gfCNCPoint3[19161] = {X 213.4015, Y 92.7444, Z -4.6667, A 0.000, B 0.000, C 0.000 }
gfCNCPoint3[19162] = {X 214.4547, Y 92.6556, Z -4.6667, A 0.000, B 0.000, C 0.000 }
gfCNCPoint3[19163] = {X 215.5100, Y 92.5955, Z -4.6667, A 0.000, B 0.000, C 0.000 }
gfCNCPoint3[19164] = {X 216.1640, Y 92.5235, Z -4.6667, A 0.000, B 0.000, C 0.000 }
gfCNCPoint3[19165] = {X 216.7937, Y 92.3327, Z -4.6667, A 0.000, B 0.000, C 0.000 }
gfCNCPoint3[19166] = {X 217.3778, Y 92.0297, Z -4.6667, A 0.000, B 0.000, C 0.000 }
gfCNCPoint3[19167] = {X 222.9188, Y 88.4538, Z -4.6667, A 0.000, B 0.000, C 0.000 }
gfCNCPoint3[19168] = {X 245.6528, Y 73.9167, Z -4.6667, A 0.000, B 0.000, C 0.000 }
gfCNCPoint3[19169] = {X 221.6008, Y 64.4780, Z -4.6667, A 0.000, B 0.000, C 0.000 }
gfCNCPoint3[19170] = {X 219.8423, Y 63.8893, Z -4.6667, A 0.000, B 0.000, C 0.000 }
gfCNCPoint3[19171] = {X 218.0279, Y 63.5055, Z -4.6667, A 0.000, B 0.000, C 0.000 }
gfCNCPoint3[19172] = {X 216.1816, Y 63.3315, Z -4.6667, A 0.000, B 0.000, C 0.000 }
gfCNCPoint3[19173] = {X 215.2274, Y 63.1935, Z -4.6667, A 0.000, B 0.000, C 0.000 }
gfCNCPoint3[19174] = {X 214.3262, Y 62.8509, Z -4.6667, A 0.000, B 0.000, C 0.000 }
gfCNCPoint3[19175] = {X 213.5213, Y 62.3203, Z -4.6667, A 0.000, B 0.000, C 0.000 }
gfCNCPoint3[19176] = {X 212.8512, Y 61.6271, Z -4.6667, A 0.000, B 0.000, C 0.000 }
gfCNCPoint3[19177] = {X 212.3482, Y 60.8046, Z -4.6667, A 0.000, B 0.000, C 0.000 }
gfCNCPoint3[19178] = {X 212.0364, Y 59.8923, Z -4.6667, A 0.000, B 0.000, C 0.000 }
gfCNCPoint3[19179] = {X 211.9308, Y 58.9341, Z -4.6667, A 0.000, B 0.000, C 0.000 }
gfCNCPoint3[19180] = {X 211.9308, Y 58.0000, Z -4.6667, A 0.000, B 0.000, C 0.000 }
gfCNCPoint3[19181] = {X 212.0411, Y 57.0209, Z -4.6667, A 0.000, B 0.000, C 0.000 }
gfCNCPoint3[19182] = {X 212.3665, Y 56.0909, Z -4.6667, A 0.000, B 0.000, C 0.000 }
gfCNCPoint3[19183] = {X 212.8907, Y 55.2566, Z -4.6667, A 0.000, B 0.000, C 0.000 }
gfCNCPoint3[19184] = {X 213.5875, Y 54.5599, Z -4.6667, A 0.000, B 0.000, C 0.000 }
gfCNCPoint3[19185] = {X 214.4217, Y 54.0357, Z -4.6667, A 0.000, B 0.000, C 0.000 }
gfCNCPoint3[19186] = {X 215.3517, Y 53.7103, Z -4.6667, A 0.000, B 0.000, C 0.000 }
gfCNCPoint3[19187] = {X 216.3308, Y 53.6000, Z -4.6667, A 0.000, B 0.000, C 0.000 }
gfCNCPoint3[19188] = {X 237.2617, Y 53.6000, Z -4.6667, A 0.000, B 0.000, C 0.000 }
gfCNCPoint3[19189] = {X 238.2408, Y 53.7103, Z -4.6667, A 0.000, B 0.000, C 0.000 }
gfCNCPoint3[19190] = {X 239.1708, Y 54.0357, Z -4.6667, A 0.000, B 0.000, C 0.000 }
gfCNCPoint3[19191] = {X 240.0050, Y 54.5599, Z -4.6667, A 0.000, B 0.000, C 0.000 }
gfCNCPoint3[19192] = {X 240.7017, Y 55.2566, Z -4.6667, A 0.000, B 0.000, C 0.000 }
gfCNCPoint3[19193] = {X 241.2260, Y 56.0909, Z -4.6667, A 0.000, B 0.000, C 0.000 }
gfCNCPoint3[19194] = {X 241.5514, Y 57.0209, Z -4.6667, A 0.000, B 0.000, C 0.000 }
gfCNCPoint3[19195] = {X 241.6617, Y 58.0000, Z -4.6667, A 0.000, B 0.000, C 0.000 }
gfCNCPoint3[19196] = {X 241.6617, Y 58.1776, Z -4.6667, A 0.000, B 0.000, C 0.000 }
gfCNCPoint3[19197] = {X 248.1442, Y 60.7053, Z -4.6667, A 0.000, B 0.000, C 0.000 }
gfCNCPoint3[19198] = {X 275.5528, Y 71.5843, Z -4.6667, A 0.000, B 0.000, C 0.000 }
gfCNCPoint3[19199] = {X 275.5523, Y 63.2811, Z -4.6667, A 0.000, B 0.000, C 0.000 }
gfCNCPoint3[19200] = {X 274.6931, Y 63.0559, Z -4.6667, A 0.000, B 0.000, C 0.000 }
gfCNCPoint3[19201] = {X 273.8966, Y 62.6627, Z -4.6667, A 0.000, B 0.000, C 0.000 }
gfCNCPoint3[19202] = {X 273.1953, Y 62.1175, Z -4.6667, A 0.000, B 0.000, C 0.000 }
gfCNCPoint3[19203] = {X 272.6178, Y 61.4426, Z -4.6667, A 0.000, B 0.000, C 0.000 }
gfCNCPoint3[19204] = {X 272.1877, Y 60.6655, Z -4.6667, A 0.000, B 0.000, C 0.000 }
gfCNCPoint3[19205] = {X 271.9223, Y 59.8178, Z -4.6667, A 0.000, B 0.000, C 0.000 }
gfCNCPoint3[19206] = {X 271.8327, Y 58.9341, Z -4.6667, A 0.000, B 0.000, C 0.000 }
gfCNCPoint3[19207] = {X 271.8327, Y 58.0000, Z -4.6667, A 0.000, B 0.000, C 0.000 }
gfCNCPoint3[19208] = {X 271.9430, Y 57.0209, Z -4.6667, A 0.000, B 0.000, C 0.000 }
gfCNCPoint3[19209] = {X 272.2684, Y 56.0909, Z -4.6667, A 0.000, B 0.000, C 0.000 }
gfCNCPoint3[19210] = {X 272.7926, Y 55.2566, Z -4.6667, A 0.000, B 0.000, C 0.000 }
gfCNCPoint3[19211] = {X 273.4893, Y 54.5599, Z -4.6667, A 0.000, B 0.000, C 0.000 }
gfCNCPoint3[19212] = {X 274.3236, Y 54.0357, Z -4.6667, A 0.000, B 0.000, C 0.000 }
gfCNCPoint3[19213] = {X 275.2536, Y 53.7103, Z -4.6667, A 0.000, B 0.000, C 0.000 }
gfCNCPoint3[19214] = {X 276.2327, Y 53.6000, Z -4.6667, A 0.000, B 0.000, C 0.000 }
gfCNCPoint3[19215] = {X 292.7731, Y 53.6000, Z -4.6667, A 0.000, B 0.000, C 0.000 }
gfCNCPoint3[19216] = {X 293.7522, Y 53.7103, Z -4.6667, A 0.000, B 0.000, C 0.000 }
gfCNCPoint3[19217] = {X 294.6822, Y 54.0357, Z -4.6667, A 0.000, B 0.000, C 0.000 }
gfCNCPoint3[19218] = {X 295.5164, Y 54.5599, Z -4.6667, A 0.000, B 0.000, C 0.000 }
gfCNCPoint3[19219] = {X 296.2131, Y 55.2566, Z -4.6667, A 0.000, B 0.000, C 0.000 }
gfCNCPoint3[19220] = {X 296.7373, Y 56.0909, Z -4.6667, A 0.000, B 0.000, C 0.000 }
gfCNCPoint3[19221] = {X 297.0628, Y 57.0209, Z -4.6667, A 0.000, B 0.000, C 0.000 }
gfCNCPoint3[19222] = {X 297.1731, Y 58.0000, Z -4.6667, A 0.000, B 0.000, C 0.000 }
gfCNCPoint3[19223] = {X 297.1731, Y 58.9353, Z -4.6667, A 0.000, B 0.000, C 0.000 }
gfCNCPoint3[19224] = {X 297.0811, Y 59.8183, Z -4.6667, A 0.000, B 0.000, C 0.000 }
gfCNCPoint3[19225] = {X 296.8144, Y 60.6650, Z -4.6667, A 0.000, B 0.000, C 0.000 }
